	160:
		IF NOT DP_SinStepe THEN	
				IF arrAxisCtrl[AxiseNo.AxisName.AnDTCarryingUpDown].Status.Homed AND arrAxisCtrl[AxiseNo.AxisName.AnDTCarryingUpDown].Status.NoMoving AND 
					NOT arrAxisCtrl[AxiseNo.AxisName.AnDTCarryingUpDown].Status.Error AND arrAxisCtrl[AxiseNo.AxisName.AnDTCarryingLine].Cmd.arrbRealPoint[1] THEN
							IF arrAxisCtrl[AxiseNo.AxisName.AnDTCarryingUpDown].Cmd.arrbRealPoint[2] THEN
								arrAxisCtrl[AxiseNo.AxisName.AnDTCarryingUpDown].Cmd.iGoSetPos:=0;
							ELSE
								arrAxisCtrl[AxiseNo.AxisName.AnDTCarryingUpDown].Cmd.iGoSetPos:=2;//正极叠片平台升降去取片位 放片
							END_IF
				END_IF
				IF 	arrAxisCtrl[AxiseNo.AxisName.AnDTCarryingUpDown].Cmd.arrbRealPoint[2] AND arrAxisCtrl[AxiseNo.AxisName.AnDTCarryingUpDown].Status.Homed THEN
								IF Mach_Control.DT_b.SinStepMode THEN//单步调试模式
									DP_SinStepe:=TRUE;
								ELSE
									DP_SinStepe:=FALSE;	
								END_IF				
								An_Step2:=170;
				END_IF	
		END_IF
	
	170:

			arrCyCtrl[arrCyNo.ElectValveName.AnDTCarryingVacuum].Cmd.bOFF:=FALSE;//正极叠片搬运真空关
			arrCyCtrl[arrCyNo.ElectValveName.AnDTCarryingVacuum].Cmd.bON:=TRUE;//正极叠片搬运真空关
			arrCyCtrl[arrCyNo.ElectValveName.AnDTCarryingVacuumBark].Cmd.bON:=TRUE;//正极叠片搬运破真空开
			arrCyCtrl[arrCyNo.ElectValveName.AnDTCarryingVacuumBark].Cmd.bOFF:=FALSE;//正极叠片搬运破真空开
			arrCyCtrl[arrCyNo.ElectValveName.AndeviationVacuum].Cmd.bON:=TRUE;//正极纠偏平台真空开		
			arrCyCtrl[arrCyNo.ElectValveName.AndeviationVacuum].Cmd.bOFF:=FALSE;//正极纠偏平台真空开	
			//IF Mach_Control.An_b.An_DPCarryingFalg THEN	
				Mach_Control.An_b.An_DPCarryingFalg :=FALSE;//复位正极叠片搬运吸盘上有料标记
				Mach_Control.An_b.An_deviationFalg:=TRUE;//置位纠偏平台上有料标记
			//END_IF
			An_Step2:=180;

			
	180:
		IF NOT DP_SinStepe THEN	
				IF arrAxisCtrl[AxiseNo.AxisName.AnDTCarryingUpDown].Status.Homed AND arrAxisCtrl[AxiseNo.AxisName.AnDTCarryingUpDown].Status.NoMoving AND 
					NOT arrAxisCtrl[AxiseNo.AxisName.AnDTCarryingUpDown].Status.Error AND arrAxisCtrl[AxiseNo.AxisName.AnDTCarryingLine].Cmd.arrbRealPoint[1] THEN
							IF arrAxisCtrl[AxiseNo.AxisName.AnDTCarryingUpDown].Cmd.arrbRealPoint[4] THEN
								arrAxisCtrl[AxiseNo.AxisName.AnDTCarryingUpDown].Cmd.iGoSetPos:=0;
							ELSE
								arrAxisCtrl[AxiseNo.AxisName.AnDTCarryingUpDown].Cmd.iGoSetPos:=4;//正极叠片平台升降去等待位
							END_IF
				END_IF
				IF 	arrAxisCtrl[AxiseNo.AxisName.AnDTCarryingUpDown].Cmd.arrbRealPoint[4] AND arrAxisCtrl[AxiseNo.AxisName.AnDTCarryingUpDown].Status.Homed THEN
								IF Mach_Control.DT_b.SinStepMode THEN//单步调试模式
									DP_SinStepe:=TRUE;
								ELSE
									DP_SinStepe:=FALSE;	
								END_IF				
								An_Step2:=190;
				END_IF	
		END_IF	
	190:
			YS.IN:=TRUE;
			
		IF 	 (Mach_Control.An_b.RectifydevDone OR CCD.AnRec.Finish.RectifyResult=2 OR CCD.AnRec.Finish.RectifyResult=3 OR CCD.AnRec.Finish.RectifyResult=4) AND YS.Q  THEN
			Mach_Control.An_b.An_Rectifydev_CS:=Mach_Control.An_b.An_Rectifydev_CS+1;
			An_Step2:=200;
			YS.IN:=FALSE;
		END_IF
		
	200:
		IF NOT DP_SinStepe THEN	
				IF arrAxisCtrl[AxiseNo.AxisName.AnDTCarryingUpDown].Status.Homed AND arrAxisCtrl[AxiseNo.AxisName.AnDTCarryingUpDown].Status.NoMoving AND 
					NOT arrAxisCtrl[AxiseNo.AxisName.AnDTCarryingUpDown].Status.Error AND arrAxisCtrl[AxiseNo.AxisName.AnDTCarryingLine].Cmd.arrbRealPoint[1] THEN
							IF arrAxisCtrl[AxiseNo.AxisName.AnDTCarryingUpDown].Cmd.arrbRealPoint[2] THEN
								arrAxisCtrl[AxiseNo.AxisName.AnDTCarryingUpDown].Cmd.iGoSetPos:=0;
							ELSE
								arrAxisCtrl[AxiseNo.AxisName.AnDTCarryingUpDown].Cmd.iGoSetPos:=2;//正极叠片平台升降去取片位 放片
							END_IF
				END_IF
				IF 	arrAxisCtrl[AxiseNo.AxisName.AnDTCarryingUpDown].Cmd.arrbRealPoint[2] AND arrAxisCtrl[AxiseNo.AxisName.AnDTCarryingUpDown].Status.Homed THEN
								IF Mach_Control.DT_b.SinStepMode THEN//单步调试模式
									DP_SinStepe:=TRUE;
								ELSE
									DP_SinStepe:=FALSE;	
								END_IF				
								An_Step2:=220;
								IF Mach_Control.DT_b.DT_CCD_TwoModel THEN												
										CCD.AnRec.Finish.RectifyResult:=0;
										CCD.AnRec.Finish.RectifyX1:=0;
										CCD.AnRec.Finish.RectifyX2:=0;
										CCD.AnRec.Finish.RectifyY:=0;												
										Mach_Control.An_b.An_CCDStart :=TRUE;//启动CCD拍照
										CCD.AnRec.Start.iPhotoDo:=2;//第二次拍照		
								END_IF	
				END_IF	
		END_IF	
		
			
	220:
	
			arrCyCtrl[arrCyNo.ElectValveName.AnDTCarryingVacuum].Cmd.bON:=FALSE;//正极叠片搬运真空开
			arrCyCtrl[arrCyNo.ElectValveName.AnDTCarryingVacuum].Cmd.bOFF:=TRUE;//正极叠片搬运真空开
			arrCyCtrl[arrCyNo.ElectValveName.AnDTCarryingVacuumBark].Cmd.bOFF:=TRUE;//正极叠片搬运破真空关
			arrCyCtrl[arrCyNo.ElectValveName.AnDTCarryingVacuumBark].Cmd.bON:=FALSE;//正极叠片搬运破真空关
			arrCyCtrl[arrCyNo.ElectValveName.AndeviationVacuum].Cmd.bOFF:=TRUE;//正极纠偏平台真空关	
			arrCyCtrl[arrCyNo.ElectValveName.AndeviationVacuum].Cmd.bON:=FALSE;//正极纠偏平台真空关	
			arrCyCtrl[arrCyNo.ElectValveName.AndeviationVacuumBark].Cmd.bON:=TRUE;//正极纠偏平台破真空开	
			arrCyCtrl[arrCyNo.ElectValveName.AndeviationVacuumBark].Cmd.bOFF:=FALSE;//正极纠偏平台破真空开	
			//IF Mach_Control.An_b.An_deviationFalg THEN
				Mach_Control.An_b.An_DPCarryingFalg :=TRUE;//叠片搬运吸盘上有料标记
				Mach_Control.An_b.An_deviationFalg:=FALSE;//纠偏平台上有料标记
			//END_IF
			YS1.IN:=TRUE;
			IF YS1.Q THEN
			An_Step2:=230;
			YS1.IN:=FALSE;
			END_IF
	
	
	230:
		IF NOT DP_SinStepe THEN	
				IF arrAxisCtrl[AxiseNo.AxisName.AnDTCarryingUpDown].Status.Homed AND arrAxisCtrl[AxiseNo.AxisName.AnDTCarryingUpDown].Status.NoMoving AND 
					NOT arrAxisCtrl[AxiseNo.AxisName.AnDTCarryingUpDown].Status.Error AND arrAxisCtrl[AxiseNo.AxisName.AnDTCarryingLine].Cmd.arrbRealPoint[1] THEN
							IF arrAxisCtrl[AxiseNo.AxisName.AnDTCarryingUpDown].Cmd.arrbRealPoint[4] THEN
								arrAxisCtrl[AxiseNo.AxisName.AnDTCarryingUpDown].Cmd.iGoSetPos:=0;
							ELSE
								arrAxisCtrl[AxiseNo.AxisName.AnDTCarryingUpDown].Cmd.iGoSetPos:=4;//正极叠片平台升降去等待位
							END_IF
				END_IF
				IF 	arrAxisCtrl[AxiseNo.AxisName.AnDTCarryingUpDown].Cmd.arrbRealPoint[4] AND arrAxisCtrl[AxiseNo.AxisName.AnDTCarryingUpDown].Status.Homed THEN
								IF Mach_Control.DT_b.SinStepMode THEN//单步调试模式
									DP_SinStepe:=TRUE;
								ELSE
									DP_SinStepe:=FALSE;	
								END_IF				
								An_Step2:=6666;
				END_IF	
		END_IF	
	
	
		
			
		
		
END_CASE
END_IF
END_ACTION

ACTION An_StandbySub4:
IF Mach_Control.U.DT_iMode=1 THEN//在自动状态下	
//An_Step3----正极叠片搬运取纠偏极片
CASE An_Step3 OF
	10://正极NG料盒气缸伸出	
		IF  arrAxisCtrl[AxiseNo.AxisName.AnDTCarryingUpDown].Status.Enabled AND  arrAxisCtrl[AxiseNo.AxisName.AnDTCarryingLine].Status.Enabled THEN	
			arrCyCtrl[arrCyNo.CylinderName.AnScrapbinCy].Cmd.bON:=TRUE;//正极纠偏气缸伸出
			IF  arrCyCtrl[arrCyNo.CylinderName.AnScrapbinCy].Status.ONState THEN
				An_Step3:=11;
			END_IF
		END_IF
	11://正极叠片搬运升降至等待位		
					IF NOT DP_SinStepe THEN	
						(*
						IF arrAxisCtrl[AxiseNo.AxisName.AnCarryingUpDown].Status.Homed AND arrAxisCtrl[AxiseNo.AxisName.AnCarryingUpDown].Status.NoMoving AND 
							NOT arrAxisCtrl[AxiseNo.AxisName.AnCarryingUpDown].Status.Error THEN
									IF arrAxisCtrl[AxiseNo.AxisName.AnCarryingUpDown].Cmd.arrbRealPoint[4] THEN
										arrAxisCtrl[AxiseNo.AxisName.AnCarryingUpDown].Cmd.iGoSetPos:=0;
									ELSE
										arrAxisCtrl[AxiseNo.AxisName.AnCarryingUpDown].Cmd.iGoSetPos:=4;//正极送片搬运升降等待高度
									END_IF
						END_IF
						*)
						IF arrAxisCtrl[AxiseNo.AxisName.AnDTCarryingUpDown].Status.Homed AND arrAxisCtrl[AxiseNo.AxisName.AnDTCarryingUpDown].Status.NoMoving AND 
							NOT arrAxisCtrl[AxiseNo.AxisName.AnDTCarryingUpDown].Status.Error THEN
									IF arrAxisCtrl[AxiseNo.AxisName.AnDTCarryingUpDown].Cmd.arrbRealPoint[4] THEN
										arrAxisCtrl[AxiseNo.AxisName.AnDTCarryingUpDown].Cmd.iGoSetPos:=0;
									ELSE
										arrAxisCtrl[AxiseNo.AxisName.AnDTCarryingUpDown].Cmd.iGoSetPos:=4;//正极叠片平台升降至等待高度
									END_IF
						END_IF
						IF 	arrAxisCtrl[AxiseNo.AxisName.AnDTCarryingUpDown].Cmd.arrbRealPoint[4] AND arrAxisCtrl[AxiseNo.AxisName.AnDTCarryingUpDown].Status.Homed THEN
										IF Mach_Control.DT_b.SinStepMode THEN//单步调试模式
											DP_SinStepe:=TRUE;
										ELSE
											DP_SinStepe:=FALSE;	
										END_IF				
										An_Step3:=30;
						END_IF	
				END_IF								
	20://正极搬运平移回初始位
		IF NOT DP_SinStepe THEN
				IF arrAxisCtrl[AxiseNo.AxisName.AnCarryingUpDown].Cmd.arrbRealPoint[4] AND arrAxisCtrl[AxiseNo.AxisName.AnCarryingLine].Status.Homed AND
					 arrAxisCtrl[AxiseNo.AxisName.AnCarryingLine].Status.NoMoving AND NOT arrAxisCtrl[AxiseNo.AxisName.AnCarryingLine].Status.Error THEN
							IF arrAxisCtrl[AxiseNo.AxisName.AnCarryingLine].Cmd.arrbRealPoint[1] THEN
									An_CarryingTorMark:=FALSE;//正极搬运1移位力矩判断标志位
									arrAxisCtrl[AxiseNo.AxisName.AnCarryingLine].Cmd.iGoSetPos:=0;
									IF Mach_Control.DT_b.SinStepMode THEN//单步调试模式
										DP_SinStepe:=TRUE;
									ELSE
										DP_SinStepe:=FALSE;	
									END_IF	
									An_Step3:=30;
							ELSE
								arrAxisCtrl[AxiseNo.AxisName.AnCarryingLine].Cmd.iGoSetPos:=1;//正极搬运平移到初始位
								An_CarryingTorMark:=TRUE;//正极搬运1移位力矩判断标志位
							END_IF
				END_IF	
		END_IF
	30://正极叠片搬运平移至初始位，
			//IF arrAxisCtrl[AxiseNo.AxisName.AnDTCarryingLine].Status.fActPos < (arrAxisPar[AxiseNo.AxisName.AnDTCarryingLine].arrTargetPoint[2]-180) THEN
	          //arrCyCtrl[arrCyNo.ElectValveName.AndeviationIonizedWind].Cmd.bON:=TRUE;//正极纠偏平台除尘
			   //arrCyCtrl[arrCyNo.ElectValveName.AndeviationIonizedWind].Cmd.bOff:=FALSE;//正极纠偏平台除尘
	      // END_IF
			IF NOT DP_SinStepe THEN
						arrCyCtrl[arrCyNo.CylinderName.AnScrapbinCy].Cmd.bON:=TRUE;//正极纠偏气缸伸出
						IF   arrAxisCtrl[AxiseNo.AxisName.AnDTCarryingUpDown].Cmd.arrbRealPoint[4] AND arrAxisCtrl[AxiseNo.AxisName.AnDTCarryingLine].Status.Homed AND
							 arrAxisCtrl[AxiseNo.AxisName.AnDTCarryingLine].Status.NoMoving AND NOT arrAxisCtrl[AxiseNo.AxisName.AnDTCarryingLine].Status.Error  AND 
							 NOT arrAxisCtrl[AxiseNo.AxisName.AnCarryingLine].Status.Error 
                             AND LREAL_TO_REAL(arrAxisCtrl[AxiseNo.AxisName.AnCarryingLine].Status.fActPos) < (arrAxisPar[AxiseNo.AxisName.AnCarryingLine].arrTargetPoint[2]-50) AND
							 arrCyCtrl[arrCyNo.CylinderName.AnScrapbinCy].Status.ONState THEN
									IF arrAxisCtrl[AxiseNo.AxisName.AnDTCarryingLine].Cmd.arrbRealPoint[1] THEN
										An_DTCarryingTorMark:=FALSE;//正极叠台搬运力矩判断标志位
										arrAxisCtrl[AxiseNo.AxisName.AnDTCarryingLine].Cmd.iGoSetPos:=0;
										IF Mach_Control.DT_b.SinStepMode THEN//单步调试模式
											DP_SinStepe:=TRUE;
										ELSE
											DP_SinStepe:=FALSE;	
										END_IF								
										An_Step3:=40;
									ELSE
										arrAxisCtrl[AxiseNo.AxisName.AnDTCarryingLine].Cmd.iGoSetPos:=1;//正极叠片平移移动至初始位
										An_DTCarryingTorMark:=TRUE;//正极叠台搬运力矩判断标志位
									END_IF
						END_IF
			END_IF
	40://判断纠偏平台是否允许取极片
			IF NOT DP_SinStepe THEN
					IF Mach_Control.An_b.An_deviationDPOK OR Mach_Control.U.EmptyRunMode THEN
						IF Mach_Control.DT_b.SinStepMode THEN//单步调试模式
							DP_SinStepe:=TRUE;
						ELSE
							DP_SinStepe:=FALSE;	
						END_IF			
					//	CCD正极纠偏平台二次拍照-------------复检拍照
						IF Mach_Control.DT_b.DT_CCD_TwoModel THEN												
							CCD.AnRec.Finish.RectifyResult:=0;
							CCD.AnRec.Finish.RectifyX1:=0;
							CCD.AnRec.Finish.RectifyX2:=0;
							CCD.AnRec.Finish.RectifyY:=0;												
							Mach_Control.An_b.An_CCDStart :=TRUE;//启动CCD拍照
							CCD.AnRec.Start.iPhotoDo:=2;//第二次拍照		
						END_IF	
						An_TON[6].IN:=FALSE;
						An_Step3:=50;
					END_IF
			END_IF
END_CASE
END_IF


CASE An_Step3 OF
	50://AND arrCyCtrl[arrCyNo.CylinderName.AnScrapbinCy].Io.DIOnSwitch
		IF NOT DP_SinStepe THEN
			arrCyCtrl[arrCyNo.ElectValveName.AnDTCarryingVacuum].Cmd.bON:=FALSE;//正极叠片搬运升降真空开
			arrCyCtrl[arrCyNo.ElectValveName.AnDTCarryingVacuum].Cmd.bOFF:=TRUE;//正极叠片搬运真空开
			IF arrAxisCtrl[AxiseNo.AxisName.AnDTCarryingUpDown].Status.Homed AND arrAxisCtrl[AxiseNo.AxisName.AnDTCarryingUpDown].Status.NoMoving AND 
			NOT arrAxisCtrl[AxiseNo.AxisName.AnDTCarryingUpDown].Status.Error  THEN
				IF arrAxisCtrl[AxiseNo.AxisName.AnDTCarryingUpDown].Cmd.arrbRealPoint[2] THEN
					arrCyCtrl[arrCyNo.ElectValveName.AndeviationVacuum].Cmd.bOFF:=TRUE;//正极纠偏真空关
					arrCyCtrl[arrCyNo.ElectValveName.AndeviationVacuum].Cmd.bON:=FALSE;//正极纠偏真空关
					arrCyCtrl[arrCyNo.ElectValveName.AndeviationVacuumBark].Cmd.bON:=TRUE;//正极纠偏破真空开
					arrCyCtrl[arrCyNo.ElectValveName.AndeviationVacuumBark].Cmd.bOFF:=FALSE;//正极纠偏破真空开
					arrAxisCtrl[AxiseNo.AxisName.AnDTCarryingUpDown].Cmd.iGoSetPos:=0;
					//IF Mach_Control.An_b.An_deviationFalg THEN
						Mach_Control.An_b.An_DPCarryingFalg:=TRUE;// 复位正极叠片搬运真空吸盘标记有料
						Mach_Control.An_b.An_deviationFalg:=FALSE;//复位正极纠偏平台有料标记	
					//END_IF
					Par.stDT_date.An_MQ_Slice[2]:=Par.stDT_date.An_MQ_Slice[1];												
																
					IF NOT An_TON[6].Q THEN
						An_TON[6].IN:=TRUE;
					ELSE
						IF Mach_Control.DT_b.SinStepMode THEN//单步调试模式
							DP_SinStepe:=TRUE;
						ELSE
							DP_SinStepe:=FALSE;	
						END_IF		
						An_TON[6].IN:=FALSE;				
						An_Step3:=60;											
					END_IF									
				ELSE
					arrAxisCtrl[AxiseNo.AxisName.AnDTCarryingUpDown].Cmd.iGoSetPos:=2;//正极叠片平台升降下降至取料高度
				END_IF
			
			END_IF	
		END_IF
	60://正极叠片搬运升降上升至初始位
		IF arrAxisCtrl[AxiseNo.AxisName.AnDTCarryingUpDown].Status.Homed AND arrAxisCtrl[AxiseNo.AxisName.AnDTCarryingUpDown].Status.NoMoving AND 
		NOT arrAxisCtrl[AxiseNo.AxisName.AnDTCarryingUpDown].Status.Error THEN
			IF arrAxisCtrl[AxiseNo.AxisName.AnDTCarryingUpDown].Cmd.arrbRealPoint[4] THEN
				arrAxisCtrl[AxiseNo.AxisName.AnDTCarryingUpDown].Cmd.iGoSetPos:=0;
				An_Step3:=6666;
			ELSE
				arrAxisCtrl[AxiseNo.AxisName.AnDTCarryingUpDown].Cmd.iGoSetPos:=4;//正极叠片平台升降上升至初始位
			END_IF
		END_IF		
END_CASE
END_ACTION

ACTION Ca_Alarm:
//报警延时时间
Ca_AlarmTON[1](IN:= , PT:=T#80MS , Q=> , ET=> );//负极取流水线搬运升降机械手吸盘误吸极片报警延时
Ca_AlarmTON[2](IN:= , PT:=T#80MS , Q=> , ET=> );//负极取流水线搬运升降机械手吸盘掉片报警延时
Ca_AlarmTON[3](IN:= , PT:=T#80MS , Q=> , ET=> );///负极送片搬运升降机械手误吸极片报警延时
Ca_AlarmTON[4](IN:= , PT:=T#80MS , Q=> , ET=> );////负极取流水线搬运升降机械手吸盘掉片	报警延时
Ca_AlarmTON[5](IN:= , PT:=T#80MS , Q=> , ET=> );///负极叠台搬运升降机械手误吸极片报警延时
Ca_AlarmTON[6](IN:= , PT:=T#80MS , Q=> , ET=> );////负极叠台搬运升降机械手吸盘掉片报警延时
Ca_AlarmTON[7](IN:= , PT:=T#80MS , Q=> , ET=> );///负极纠偏平台误吸极片报警延时
Ca_AlarmTON[8](IN:= , PT:=T#150MS , Q=> , ET=> );////负极纠偏平台吸盘掉片报警延时
Ca_AlarmTON[9](IN:= , PT:=T#300MS , Q=> , ET=> );
Ca_AlarmTON[10](IN:= , PT:=T#300MS , Q=> , ET=> );
Ca_AlarmTON[11](IN:= , PT:=T#300MS , Q=> , ET=> );//负极极片对齐度检测返回结果超时
Ca_AlarmTon[12](IN:= , PT:=T#400MS , Q=> , ET=> );//负极CCD纠偏平台检测返回结果超时
Ca_AlarmTon[13](IN:=CaCCDMark , PT:=T#50MS , Q=> , ET=> );//负极CCD纠偏平台检测返回结果超时
Ca_AlarmTon[15](IN:= , PT:=T#50MS , Q=> , ET=> );//负极取片搬运叠片过程中的真空处理
Ca_AlarmTon[16](IN:= , PT:=T#50MS , Q=> , ET=> );//负极取片搬运叠片过程中的真空处理
Ca_AlarmTon[17](IN:=NOT Mach_Control.se.CaNGboxsensor , PT:=T#5S , Q=> , ET=> );//负极NG料盒料满	

rCaUse[1](CLK:=Ca_Step0=40, Q=> );
rCaUse[2](CLK:=Mach_Control.Ca_b.Ca_CCDStart AND NOT   Mach_Control.Ca_b.Demarcateing , Q=> );
rCaUse[3](CLK:=Par.stDT_date.Ca_Rectifydev_Btn , Q=> );
rCaUse[4](CLK:= NOT arrCyCtrl[arrCyNo.ElectValveName.CaCarryingVacuum2].Io.DOStatus1 , Q=> ); 
rCaUse[5](CLK:= NOT arrCyCtrl[arrCyNo.ElectValveName.CaDTCarryingVacuum].Io.DOStatus1 , Q=> );
rCaUse[6](CLK:=arrCyCtrl[arrCyNo.ElectValveName.CaCarryingVacuum1].Io.DOStatus1 , Q=> ); 

//Mach_Control.Ca_b.Error[1]:=TRUE;//负极取流水线搬运升降有真空信号，无极片报警
//Mach_Control.Ca_b.Error[2]:=TRUE;//负极取流水线搬运升降有极片，无真空信号报警
//Mach_Control.Ca_b.Error[3]:=TRUE;//负极送片搬运升降有真空信号，无极片报警
//Mach_Control.Ca_b.Error[4]:=TRUE;//负极送片搬运升降取片过程中真空报警,有极片，无真空信号
//Mach_Control.Ca_b.Error[5]:=TRUE;//负极叠台搬运升降有真空信号，无极片报警
//Mach_Control.Ca_b.Error[6]:=TRUE;//负极叠台搬运升降有极片，无真空信号报警
//Mach_Control.Ca_b.Error[7]:=TRUE;//纠偏平台无片极，有真空信号报警
//Mach_Control.Ca_b.Error[8]:=TRUE;//纠偏平台有极片，无真空报警
//Mach_Control.Ca_b.Error[9]:=TRUE;//纠偏CCD拍照完成IO信号未给出
//Mach_Control.Ca_b.Error[10] //CCD标定NG报警
//Mach_Control.Ca_b.Error[11]:=TRUE;//负极藕合凸轮报警
//Mach_Control.Ca_b.Error[12]:=TRUE;//负极NG收纳盒满料报警
//Mach_Control.Ca_b.Error[13];
//Mach_Control.Ca_b.Error[14];
//Mach_Control.Ca_b.Error[15];
//Mach_Control.Ca_b.Error[16];
//Mach_Control.Ca_b.Error[17]:=TRUE;//负极防撞感应信报警
//Mach_Control.Ca_b.Error[18] :=TRUE;//负极CCD纠偏平台检测返回结果超时
//Mach_Control.Ca_b.Error[19]:=TRUE;//负极取放料回原点超时报警
//Mach_Control.Ca_b.Error[20]:=TRUE;//负极皮带回原点超时报警	
//Mach_Control.Ca_b.Error[21]:=TRUE;//负极纠偏平台连续NG报警
//Mach_Control.Ca_b.Error[22]:=TRUE;//负极叠台搬运升降真空报警，电芯上有片，请拿掉
//Mach_Control.Ca_b.Error[23]:=TRUE;//负极叠台搬运升降真空报警，电芯上无掉片
//Mach_Control.Ca_b.Error[24] //负极纠偏平台NG片未排掉报警，请拿掉
//Mach_Control.Ca_b.Error[25] //负极极片对齐度检测返回结果超时
//Mach_Control.Ca_b.Error[26]:=TRUE;//负极搬运平移防撞软限位报警
//Mach_Control.Ca_b.Error[27] ////负极极片对齐度检测返回结果无片报警
//Mach_Control.Ca_b.Error[28] //负极极片NG料盒料满
//Mach_Control.Ca_b.Error[29]:=TRUE;	  //负极初始化时负极叠片搬运升降吸盘有真空报警
//Mach_Control.Ca_b.Error[30]:=TRUE;	  //负极初始化时负极送片搬运升降2吸盘有真空报警
//Mach_Control.Ca_b.Error[31]:=TRUE;	   //负极皮带初始化时负极送片搬运升降1吸盘有真空报警


//Mach_Control.Ca_b.Error[32]:=TRUE;//负极取片叠片过程中真空报警
//Mach_Control.Ca_b.Error[33]:=TRUE;//纠偏平台有片，请拿走
//Mach_Control.Ca_b.Error[34]:=TRUE;//负极叠台搬运平移取片时真空报警
//Mach_Control.Ca_b.Error[35]:=TRUE;//负极纠偏台NG料盒料满报警
//Mach_Control.Ca_b.Error[36]:=TRUE;//负极纠偏纠偏CCD返回结果超时
//Mach_Control.Ca_b.Error[38] :=TRUE;//负极叠台搬运升降有极耳无真空报警
//Mach_Control.Ca_b.Error[39] :=TRUE;//负极叠台搬运升降有极耳无真空报警
//Mach_Control.Ca_b.Error[40] S=AnOverNGcount>=3;//负极单张踢废连续NG
//Mach_Control.Ca_b.Error[41] :=TRUE;//负极缓存皮带准备运动时，负极升降1不在安全位报警
//Mach_Control.Ca_b.Error[42] :=TRUE;//负极机械手初始化时，叠台搬运升降不在避让位
Mach_Control.Ca_b.Error[40] S=CaOverNGcount>=3;//负极单张踢废连续NG

//NG料盒料满报警
	IF (*Par.stDT_date.Ca_Rectifydev_JS>=Par.stDT_date.Ca_Rectifydev_NGSet OR*) Ca_AlarmTon[17].Q THEN
		Mach_Control.Ca_b.Error[35]:=TRUE;//负极纠偏台NG料盒料满报警
	ELSE
		Mach_Control.Ca_b.Error[35]:=FALSE;//负极纠偏台NG料盒料满报警
	END_IF
	IF rCaUse[3].Q THEN
		Par.stDT_date.Ca_Rectifydev_JS:=0;
	END_IF
	
	
	
//负极初始化时有真空报警	
	IF Mach_Control.Ca_b.Ca_GohomeHMI  THEN
			IF  arrCyCtrl[arrCyNo.ElectValveName.CaDTCarryingVacuum].Status.ONState  THEN
				Mach_Control.Ca_b.Error[29]:=TRUE;	  //负极初始化时负极叠片搬运升降吸盘有真空报警
			END_IF
			IF arrCyCtrl[arrCyNo.ElectValveName.CaCarryingVacuum2].Status.ONState THEN
				Mach_Control.Ca_b.Error[30]:=TRUE;	  //负极初始化时负极送片搬运升降2吸盘有真空报警
			END_IF
	END_IF	
//负极皮带初始化时有真空报警	
	IF Mach_Control.Ca_b.Ca_BeltGohomeHMI  AND arrCyCtrl[arrCyNo.ElectValveName.CaCarryingVacuum1].Status.ONState THEN
		Mach_Control.Ca_b.Error[31]:=TRUE;	   //负极皮带初始化时负极送片搬运升降1吸盘有真空报警
	END_IF	
	
//负极取流水线搬运机械手升降吸盘真空信号与搬运升降极片有无料标记不一致报警
Ca_AlarmTON[1].IN:=NOT arrCyCtrl[arrCyNo.ElectValveName.CaCarryingVacuum1].Io.DOStatus1 AND  arrCyCtrl[arrCyNo.ElectValveName.CaCarryingVacuum1].Io.DIOnSwitch 
	AND NOT Mach_Control.Ca_b.Ca_SegbeltFalg AND NOT Mach_Control.U.EmptyRunMode AND  Mach_Control.U.DT_iMode=1 AND NOT Mach_Control.Ca_b.Error[2] ;
rtVacALM[1](CLK:=Ca_AlarmTON[1].Q, Q=> );		
		IF  rtVacALM[1].Q THEN
			//Mach_Control.Ca_b.Ca_SegbeltFalg:=FALSE;
			Mach_Control.Ca_b.Error[1]:=TRUE;//负极取流水线搬运升降有真空信号，无极片报警
		END_IF

//
Ca_AlarmTON[2].IN:=NOT arrCyCtrl[arrCyNo.ElectValveName.CaCarryingVacuum1].Io.DIOnSwitch AND  Mach_Control.Ca_b.Ca_SegbeltFalg AND NOT Mach_Control.U.EmptyRunMode AND
	arrAxisCtrl[AxiseNo.AxisName.CaCarryingUpDown1].Status.fActPos<=(arrAxisPar[AxiseNo.AxisName.CaCarryingUpDown1].arrTargetPoint[2]-5) AND arrCyCtrl[arrCyNo.ElectValveName.CaCarryingVacuum1].Io.DOStatus1 ;		
rtVacALM[2](CLK:=Ca_AlarmTON[2].Q, Q=> );	
		IF  rtVacALM[2].Q THEN
			Mach_Control.Ca_b.Error[2]:=TRUE;//负极取流水线搬运升降有极片，无真空信号报警
		END_IF	
	
(*
//负极取流水线搬运机械手升降吸盘真空信号与搬运升降极片有无料标记不一致报警
Ca_AlarmTON[1].IN:=NOT arrCyCtrl[arrCyNo.ElectValveName.CaCarryingVacuum1].Io.DOStatus1 AND  arrCyCtrl[arrCyNo.ElectValveName.CaCarryingVacuum1].Io.DIOnSwitch 
	AND NOT Mach_Control.Ca_b.Ca_SegbeltFalg AND NOT Mach_Control.U.EmptyRunMode AND  Mach_Control.U.DT_iMode=1 AND NOT Mach_Control.Ca_b.Error[2] ;
		IF  Ca_AlarmTON[1].Q THEN
			//Mach_Control.Ca_b.Ca_SegbeltFalg:=FALSE;
			Mach_Control.Ca_b.Error[1]:=TRUE;//负极取流水线搬运升降有真空信号，无极片报警
		END_IF

//
Ca_AlarmTON[2].IN:=NOT arrCyCtrl[arrCyNo.ElectValveName.CaCarryingVacuum1].Io.DIOnSwitch AND  Mach_Control.Ca_b.Ca_SegbeltFalg AND NOT Mach_Control.U.EmptyRunMode AND
	arrAxisCtrl[AxiseNo.AxisName.CaCarryingUpDown1].Status.fActPos<=(arrAxisPar[AxiseNo.AxisName.CaCarryingUpDown1].arrTargetPoint[2]-5) AND arrCyCtrl[arrCyNo.ElectValveName.CaCarryingVacuum1].Io.DOStatus1 ;		
		IF  Ca_AlarmTON[2].Q THEN
			(*
			arrCyCtrl[arrCyNo.ElectValveName.CaCarryingVacuum1]	.Cmd.bOFF:=TRUE;//负极搬运1真空关
			arrCyCtrl[arrCyNo.ElectValveName.CaCarryingVacuum1]	.Cmd.bON:=FALSE;//负极搬运1真空开
			arrCyCtrl[arrCyNo.ElectValveName.CaCarryingVacuumBark1]	.Cmd.bOFF:=FALSE;//负极搬运1真空关
			arrCyCtrl[arrCyNo.ElectValveName.CaCarryingVacuumBark1]	.Cmd.bON:=TRUE;//负极搬运1真空开
			Mach_Control.Ca_b.Ca_SegbeltFalg:=FALSE;
			*)
			Mach_Control.Ca_b.Error[2]:=TRUE;//负极取流水线搬运升降有极片，无真空信号报警
		END_IF
IF Mach_Control.Ca_b.Error[2] AND arrCyCtrl[arrCyNo.ElectValveName.CaCarryingVacuum1].Io.DIOnSwitch AND rCa_AlarmReset.Q  THEN
	Mach_Control.Ca_b.Error[2]:=FALSE;//负极取流水线搬运升降有极片，无真空信号报警
ELSIF Mach_Control.Ca_b.Error[2] AND NOT arrCyCtrl[arrCyNo.ElectValveName.CaCarryingVacuum1].Io.DIOnSwitch AND rCa_AlarmReset.Q  THEN
	arrCyCtrl[arrCyNo.ElectValveName.CaCarryingVacuum1]	.Cmd.bOFF:=TRUE;//负极搬运1真空关
	arrCyCtrl[arrCyNo.ElectValveName.CaCarryingVacuum1]	.Cmd.bON:=FALSE;//负极搬运1真空开
	arrCyCtrl[arrCyNo.ElectValveName.CaCarryingVacuumBark1]	.Cmd.bOFF:=FALSE;//负极搬运1真空关
	arrCyCtrl[arrCyNo.ElectValveName.CaCarryingVacuumBark1]	.Cmd.bON:=TRUE;//负极搬运1真空开
	Ca_StandbyStep2:=0;
	Mach_Control.Ca_b.Ca_SegbeltFalg:=FALSE;
	Mach_Control.Ca_b.Error[2]:=FALSE;//负极取流水线搬运升降有极片，无真空信号报警
END_IF
*)		

//负极取片搬运取片过程中的真空报警处理
Ca_AlarmTON[4].IN:=NOT arrCyCtrl[arrCyNo.ElectValveName.CaCarryingVacuum2].Io.DIOnSwitch AND Mach_Control.Ca_b.Ca_CarryingFalg 
	AND NOT Mach_Control.U.EmptyRunMode AND arrAxisCtrl[AxiseNo.AxisName.CaCarryingUpDown2].Status.Homed 
	AND arrAxisCtrl[AxiseNo.AxisName.CaCarryingUpDown2].Status.fActPos<=(arrAxisPar[AxiseNo.AxisName.CaCarryingUpDown2].arrTargetPoint[2]-5)//AND NOT Blueflaging
	AND NOT  arrCyCtrl[arrCyNo.ElectValveName.CaCarryingVacuum2].Io.DOStatus1 AND NOT Bnt_Blueflaging  AND  arrAxisCtrl[AxiseNo.AxisName.CaCarryingLine2].Status.NoMoving ;
		IF  Ca_AlarmTON[4].Q THEN  
				Mach_Control.Ca_b.Error[4]:=TRUE;//负极送片搬运升降机械有极片，无真空信号报警
				(*
				Mach_Control.Ca_b.Ca_CarryingFalg :=FALSE;
				arrCyCtrl[arrCyNo.ElectValveName.CaCarryingVacuum2]	.Cmd.bON:=TRUE;//负极搬运2真空破
				arrCyCtrl[arrCyNo.ElectValveName.CaCarryingVacuum2]	.Cmd.bOFF:=FALSE;//负极搬运2真空破
				*)
		END_IF
IF Mach_Control.Ca_b.Error[4] AND arrCyCtrl[arrCyNo.ElectValveName.CaCarryingVacuum2].Io.DIOnSwitch AND rCa_AlarmReset.Q  THEN
	Mach_Control.Ca_b.Error[4]:=FALSE;//负极送片搬运升降机械有极片，无真空信号报警
ELSIF Mach_Control.Ca_b.Error[4] AND NOT arrCyCtrl[arrCyNo.ElectValveName.CaCarryingVacuum2].Io.DIOnSwitch AND rCa_AlarmReset.Q  THEN
	arrCyCtrl[arrCyNo.ElectValveName.CaCarryingVacuum2]	.Cmd.bON:=TRUE;//负极搬运2真空破
	arrCyCtrl[arrCyNo.ElectValveName.CaCarryingVacuum2]	.Cmd.bOFF:=FALSE;//负极搬运2真空破
	Ca_StandbyStep0:=0;
	Ca_Step0:=0;
	Ca_Step1:=0;
	Ca_Step2:=0;
	Ca_Step3:=0;
	Mach_Control.Ca_b.Error[4]:=FALSE;//负极送片搬运升降机械有极片，无真空信号报警
	Mach_Control.Ca_b.Ca_CarryingFalg :=FALSE;
END_IF
		
		
		
		

//负极取片搬运在叠片过程中的真空报警处理
Ca_AlarmTON[15].IN:=NOT arrCyCtrl[arrCyNo.ElectValveName.CaCarryingVacuum2].Io.DIOnSwitch AND Mach_Control.Ca_b.Ca_CarryingFalg 
	 AND  arrAxisCtrl[AxiseNo.AxisName.CaCarryingLine2].Status.Moving AND NOT Mach_Control.U.EmptyRunMode
	AND NOT  arrCyCtrl[arrCyNo.ElectValveName.CaCarryingVacuum2].Io.DOStatus1 AND NOT Bnt_Blueflaging
	AND  arrAxisCtrl[AxiseNo.VirAxisName.VirMain].Status.fActPos>1  AND  arrAxisCtrl[AxiseNo.VirAxisName.VirMain].Status.fActPos<232 ;
	
	IF  Ca_AlarmTON[15].Q THEN  
		CCD.CaRec.Finish.RectifyResult:=0;//拍照结果清零
		Mach_Control.Ca_b.Error[32]:=TRUE;	   //负极取片升降真空叠片过程中真空报警
		Mach_Control.Ca_b.Ca_CarryingFalg :=FALSE;
		arrCyCtrl[arrCyNo.ElectValveName.CaCarryingVacuum2]	.Cmd.bON:=TRUE;//负极搬运2真空破
		arrCyCtrl[arrCyNo.ElectValveName.CaCarryingVacuum2]	.Cmd.bOFF:=FALSE;//负极搬运2真空破
	END_IF
	//搬运平移在叠片过程中报警时，纠偏平台拍照有无片来确定是否掉片到纠偏平台
	IF Mach_Control.Ca_b.Error[32] AND rCa_AlarmReset.Q  THEN
		//CCD.CaRec.Finish.RectifyResult:=0;//拍照结果清零
		Mach_Control.Ca_b.Ca_CCDStart :=TRUE;//启动CCD拍照
		CCD.CaRec.Start.iPhotoDo:=1;//启动CCD第二次拍照
	END_IF
	IF Mach_Control.Ca_b.Error[32] AND (CCD.CaRec.Finish.RectifyResult=3  OR  Mach_Control.U.CCD_ChosesHMI) AND rCa_AlarmReset.Q  THEN
		Mach_Control.Ca_b.Error[32]:=FALSE;
		Mach_Control.Ca_b.Error[33]:=FALSE;//纠偏平台有片，请拿走
	ELSIF Mach_Control.Ca_b.Error[32] AND (CCD.CaRec.Finish.RectifyResult<>3  AND NOT   Mach_Control.U.CCD_ChosesHMI)THEN
		Mach_Control.Ca_b.Error[33]:=TRUE;//纠偏平台有片，请拿走
	END_IF
	
	

	
//负极叠片搬运升降真空信号与有无极片标记信号不一致
Ca_AlarmTON[5].IN:=(arrCyCtrl[arrCyNo.ElectValveName.CaDTCarryingVacuum].Io.DIOnSwitch OR Mach_Control.se.CaDTCarryingJROnSwitch) 
    AND NOT Mach_Control.Ca_b.Ca_DPCarryingFalg 
	AND NOT Mach_Control.U.EmptyRunMode AND Mach_Control.U.DT_iMode=1 AND iEmptyFoldStep[1]=0 AND DP_Step0<1000 AND DP_Step0>3100
	AND NOT  arrCyCtrl[arrCyNo.ElectValveName.CaDTCarryingVacuum].Io.DOStatus1  AND NOT DP_CheseCam  AND NOT Bnt_Blueflaging;//AND NOT Blueflaging
	IF  Ca_AlarmTON[5].Q THEN
		IF  arrCyCtrl[arrCyNo.ElectValveName.CaDTCarryingVacuum].Io.DIOnSwitch THEN
		   Mach_Control.Ca_b.Error[5]:=TRUE;//负极叠台搬运升降有真空信号，无极片报警
		END_IF   
		IF Mach_Control.se.CaDTCarryingJROnSwitch THEN
		   Mach_Control.Ca_b.Error[37]:=TRUE;//负极叠台搬运升降有真空信号，无极耳报警
		END_IF
	END_IF
	
//负极叠台搬运在取片过程中的真空报警处理
Ca_AlarmTON[16].IN:=(NOT arrCyCtrl[arrCyNo.ElectValveName.CaDTCarryingVacuum].Io.DIOnSwitch OR NOT Mach_Control.se.CaDTCarryingJROnSwitch) 
    AND Mach_Control.Ca_b.Ca_DPCarryingFalg AND NOT Mach_Control.U.EmptyRunMode  AND
	arrAxisCtrl[AxiseNo.AxisName.CaDTCarryingUpDown].Status.fActPos<=(arrAxisPar[AxiseNo.AxisName.CaDTCarryingUpDown].arrTargetPoint[2]-5)AND  (Ca_Step2=6666 OR Ca_Step2=0) 
	AND NOT  arrCyCtrl[arrCyNo.ElectValveName.CaDTCarryingVacuum].Io.DOStatus1 AND  arrAxisCtrl[AxiseNo.AxisName.CaDTCarryingLine].Status.NoMoving  AND iEmptyFoldStep[1]=0
	AND (DP_Step0<1000 OR DP_Step0>3100)  ;
	
	IF  Ca_AlarmTON[16].Q THEN
		//CCD.CaRec.Finish.RectifyResult:=0;//拍照结果清零
		IF   NOT arrCyCtrl[arrCyNo.ElectValveName.CaDTCarryingVacuum].Io.DIOnSwitch THEN
	    	Mach_Control.Ca_b.Error[34]:=TRUE;//负极叠台搬运升降有极片，无真空信号反馈
		END_IF		
		IF NOT Mach_Control.se.CaDTCarryingJROnSwitch THEN
		   Mach_Control.Ca_b.Error[39]:=TRUE;//负极叠台搬运升降有极耳无真空报警
		END_IF				
		Mach_Control.Ca_b.Ca_DPCarryingFalg:=FALSE;
		arrCyCtrl[arrCyNo.ElectValveName.CaDTCarryingVacuum].Cmd.bON:=TRUE;//负极叠片搬运升降真空破
		arrCyCtrl[arrCyNo.ElectValveName.CaDTCarryingVacuum].Cmd.bOFF:=FALSE;//负极叠片搬运升降真空破
	END_IF	
	//叠台搬运平移在取片过程中报警时，纠偏平台拍照有无片来确定是否掉片到纠偏平台
	IF (Mach_Control.Ca_b.Error[34] OR Mach_Control.Ca_b.Error[39]) AND rCa_AlarmReset.Q  THEN
		//CCD.CaRec.Finish.RectifyResult:=0;//拍照结果清零
		Mach_Control.Ca_b.Ca_CCDStart :=TRUE;//启动CCD拍照
		CCD.CaRec.Start.iPhotoDo:=1;//启动CCD第二次拍照
	END_IF
	IF (Mach_Control.Ca_b.Error[34]OR Mach_Control.Ca_b.Error[39]) AND (CCD.CaRec.Finish.RectifyResult=3  OR  Mach_Control.U.CCD_ChosesHMI) AND rCa_AlarmReset.Q  THEN
		Mach_Control.Ca_b.Error[34]:=FALSE;//叠台升降取片过程中真空报警，
		Mach_Control.Ca_b.Error[39]:=FALSE;//负极叠台搬运升降有极耳无真空报警
		Mach_Control.Ca_b.Error[33]:=FALSE;//纠偏平台有片，请拿走
	ELSIF (Mach_Control.Ca_b.Error[34] OR Mach_Control.Ca_b.Error[39]) AND (CCD.CaRec.Finish.RectifyResult<>3  AND NOT   Mach_Control.U.CCD_ChosesHMI)THEN
		Mach_Control.Ca_b.Error[33]:=TRUE;//纠偏平台有片，请拿走
	END_IF
	
	
	
//负极叠台搬运在叠片过程中的真空报警处理
Ca_AlarmTON[6].IN:=(NOT arrCyCtrl[arrCyNo.ElectValveName.CaDTCarryingVacuum].Io.DIOnSwitch OR NOT Mach_Control.se.CaDTCarryingJROnSwitch) 
    AND Mach_Control.Ca_b.Ca_DPCarryingFalg 
	AND NOT Mach_Control.U.EmptyRunMode  AND   (Ca_Step2=6666 OR Ca_Step2=0) 
	AND arrAxisCtrl[AxiseNo.VirAxisName.VirMain].Status.fActPos<232 AND NOT Bnt_Blueflaging  AND arrAxisCtrl[AxiseNo.VirAxisName.VirMain].Status.fActPos>1 
	AND NOT  arrCyCtrl[arrCyNo.ElectValveName.CaDTCarryingVacuum].Io.DOStatus1 AND  arrAxisCtrl[AxiseNo.VirAxisName.VirMain].Status.Moving
	AND  arrAxisCtrl[AxiseNo.AxisName.CaDTCarryingLine].Status.Moving  ;
	
	IF  Ca_AlarmTON[6].Q THEN
		//Mach_Control.DT_b.OverhandResult:=0;
		IF   NOT arrCyCtrl[arrCyNo.ElectValveName.CaDTCarryingVacuum].Io.DIOnSwitch THEN
		   Mach_Control.Ca_b.Error[6]:=TRUE;//负极叠台搬运升降有极片，无真空信号反馈
		END_IF	
		IF NOT Mach_Control.se.CaDTCarryingJROnSwitch THEN
		   Mach_Control.Ca_b.Error[38]:=TRUE;//负极叠台搬运升降有极耳无真空报警
		END_IF			
		
		Ca_Number:=TRUE;
		Mach_Control.Ca_b.Ca_DPCarryingFalg:=FALSE;
		arrCyCtrl[arrCyNo.ElectValveName.CaDTCarryingVacuum].Cmd.bON:=TRUE;//负极叠片搬运升降真空破
		arrCyCtrl[arrCyNo.ElectValveName.CaDTCarryingVacuum].Cmd.bOFF:=FALSE;//负极叠片搬运升降真空破
	END_IF	
	//负极叠台搬运升降真空报警，电芯上有片，请拿掉
	Ca_AlarmTON[9].IN:=(Mach_Control.Ca_b.Error[6] OR Mach_Control.Ca_b.Error[38] )  AND Mach_Control.DT_b.OverhandResult<>3 AND NOT Mach_Control.U.CCD_ChosesHMI  ;	
	IF  Ca_AlarmTON[9].Q THEN
		Mach_Control.Ca_b.Error[22]:=TRUE;//负极叠台搬运升降真空报警，电芯上有片，请拿掉
	END_IF
	IF fCa_AlarmRest.Q AND  Mach_Control.Ca_b.Error[22] AND arrAxisCtrl[AxiseNo.VirAxisName.VirMain].Status.fActPos<1 THEN
		CCD.Over.Start.iPhotoDo:=2;
		Mach_Control.DT_b.CDD_OverStart:=TRUE;
	END_IF 
	IF Mach_Control.Ca_b.Error[22] AND Mach_Control.DT_b.OverhandResult=3   AND rCa_AlarmReset.Q  THEN
		Mach_Control.Ca_b.Error[22]:=FALSE;//复位电芯有片报警
		Mach_Control.DT_b.OverhandResult:=0;
	END_IF	
	
	//负极叠台搬运升降真空报警，电芯上无掉片
	Ca_AlarmTON[10].IN:=(Mach_Control.Ca_b.Error[6] OR Mach_Control.Ca_b.Error[38]) AND Mach_Control.DT_b.OverhandResult=3 AND NOT Mach_Control.U.CCD_ChosesHMI    ;	
	IF  Ca_AlarmTON[10].Q THEN
			Mach_Control.Ca_b.Error[23]:=TRUE;//负极叠台搬运升降真空报警，电芯上无掉片
	END_IF	

	


	

		

//负极纠偏平台真空信号与有无料标记不一致报警
Ca_AlarmTON[7].IN:=arrCyCtrl[arrCyNo.ElectValveName.CadeviationVacuum].Io.DIOnSwitch AND NOT Mach_Control.Ca_b.Ca_deviationFalg 
	AND NOT Mach_Control.U.EmptyRunMode AND arrAxisCtrl[AxiseNo.AxisName.CaCarryingUpDown2].Status.Homed  
	AND arrAxisCtrl[AxiseNo.AxisName.CaDTCarryingUpDown].Status.fActPos<=(arrAxisPar[AxiseNo.AxisName.CaDTCarryingUpDown].arrTargetPoint[4]+5) 
	AND iEmptyFoldStep[1]=0 AND (DP_Step0<1000 OR DP_Step0>3100)   ;
		IF  Ca_AlarmTON[7].Q THEN
			Mach_Control.Ca_b.Error[7]:=TRUE;//纠偏平台无片极，有真空信号报警
		END_IF

Ca_AlarmTON[8].IN:=NOT arrCyCtrl[arrCyNo.ElectValveName.CadeviationVacuum].Io.DIOnSwitch AND Mach_Control.Ca_b.Ca_deviationFalg 
	AND NOT Mach_Control.U.EmptyRunMode AND	arrAxisCtrl[AxiseNo.AxisName.CaCarryingUpDown2].Status.Homed  
	AND arrAxisCtrl[AxiseNo.AxisName.CaCarryingUpDown2].Status.fActPos<=(arrAxisPar[AxiseNo.AxisName.CaCarryingUpDown2].arrTargetPoint[4]+5) 
	AND iEmptyFoldStep[1]=0 AND (DP_Step0<1000 OR DP_Step0>3100) AND NOT Mach_Control.Ca_b.Ca_VacuumErrorNG ;	
		IF  Ca_AlarmTON[8].Q THEN
			Mach_Control.Ca_b.Error[8]:=TRUE;//纠偏平台有极片，无真空报警
			Mach_Control.Ca_b.Ca_VacuumErrorNG:=TRUE;//负极抛真空NG料标志			
		END_IF



IF fCa_AlarmRest.Q AND  Mach_Control.Ca_b.Error[24] AND arrAxisCtrl[AxiseNo.VirAxisName.VirMain].Status.fActPos<1 THEN		
	Mach_Control.Ca_b.Ca_CCDStart :=TRUE;//启动CCD拍照
	CCD.CaRec.Start.iPhotoDo:=1;//启动CCD第二次拍照
END_IF
//负极纠偏平台片未排掉报警
IF Mach_Control.Ca_b.Error[24] AND CCD.CaRec.Finish.RectifyResult=3  AND rCa_AlarmReset.Q  THEN
	Mach_Control.Ca_b.Error[24]:=FALSE;
END_IF
//负极纠偏平台连续NG报警
IF Mach_Control.Ca_b.Ca_CCD_amount>=3 AND NOT Mach_Control.Ca_b.Error[21] THEN	
		Mach_Control.Ca_b.Error[21]:=TRUE;//负极纠偏平台连续NG报警
END_IF



//负极取料报警复位
rCa_AlarmReset(CLK:=Sys_Control.btn.System_Rrestbtn , Q=> );//负极报警复位上升沿
fCa_AlarmRest(CLK:=Sys_Control.btn.System_Rrestbtn  , Q=> );//负极报警复位下降沿
IF Mach_Control.U.DT_iMode=3 THEN//在手动状态下，复位报警
	
		IF Mach_Control.Ca_b.Error[2] AND NOT Mach_Control.Ca_b.Ca_SegbeltFalg AND rCa_AlarmReset.Q THEN
				//Mach_Control.Ca_b.Ca_SegbeltFalg:=FALSE;
				//Ca_StandbyStep2:=0;
		END_IF
		
		//IF Mach_Control.Ca_b.Error[4] AND rCa_AlarmReset.Q THEN
			//	Mach_Control.Ca_b.Ca_CarryingFalg:=FALSE;
		//END_IF
		
		IF (Mach_Control.Ca_b.Error[6] OR Mach_Control.Ca_b.Error[38]) AND rCa_AlarmReset.Q THEN
				Mach_Control.Ca_b.Ca_DPCarryingFalg:=FALSE;
		END_IF
//20240105临时屏蔽
	(*		
		IF Mach_Control.Ca_b.Error[8] AND rCa_AlarmReset.Q THEN
				 Mach_Control.Ca_b.Ca_deviationFalg:=FALSE;
		END_IF
	*)	
		IF Mach_Control.Ca_b.Error[21] AND rCa_AlarmReset.Q THEN
				 Mach_Control.Ca_b.Ca_CCD_amount:=0	;	 
		END_IF
		
		
		
																	//20240105临时屏蔽	
		IF ((Mach_Control.Ca_b.Error[4]AND NOT Mach_Control.Ca_b.Ca_CarryingFalg) OR Mach_Control.Ca_b.Error[6] OR Mach_Control.Ca_b.Error[38] ) AND rCa_AlarmReset.Q   THEN
			Ca_StandbyStep0:=0;
			Ca_Step0:=0;
			Ca_Step1:=0;
			Ca_Step2:=0;
			Ca_Step3:=0;
		END_IF
		
		//报警状态复位
		IF fCa_AlarmRest.Q AND NOT Mach_Control.Ca_b.Error[22] AND NOT Mach_Control.Ca_b.Error[4]  AND  NOT Mach_Control.Ca_b.Error[6]   
		AND NOT Mach_Control.Ca_b.Error[32] AND NOT  Mach_Control.Ca_b.Error[24] AND NOT Mach_Control.Ca_b.Error[34] 
        AND NOT  Mach_Control.Ca_b.Error[38] AND NOT  Mach_Control.Ca_b.Error[39]  THEN
			MEMSET(ADR(Mach_Control.Ca_b.Error),0,SIZEOF(Mach_Control.Ca_b.Error)); // 负极取片报警复位	
			//CaOverNGcount:=0;
			arrAxisCtrl[AxiseNo.AxisName.CaDTCarryingLine].Cmd.bStop:=FALSE;
		END_IF
		
		IF CaOverNGcount>=3 AND fCa_AlarmRest.Q  THEN
		   CaOverNGcount:=0;
		END_IF
		
		IF Mach_Control.Ca_b.Ca_DTqr AND Mach_Control.Ca_b.Error[4]   THEN
				Mach_Control.Ca_b.Error[4]:=FALSE;
				Mach_Control.Ca_b.Ca_CarryingFalg:=FALSE;
		END_IF
		
		IF Mach_Control.Ca_b.Ca_DTqr AND  (Mach_Control.Ca_b.Error[6] OR  Mach_Control.Ca_b.Error[38]) THEN
				Mach_Control.Ca_b.Error[6]:=FALSE;
				Mach_Control.Ca_b.Error[38]:=FALSE;
				Mach_Control.Ca_b.Ca_DPCarryingFalg:=FALSE;
		END_IF
		
		IF (Mach_Control.Ca_b.Error[9] OR Ca_RectifydevStep=9999) AND fCa_AlarmRest.Q THEN
				Mach_Control.Ca_b.Error[9]:=FALSE;
				Ca_RectifydevStep:=0;
				CCD.CaRec.Finish.RectifyX1:=0;
				CCD.CaRec.Finish.RectifyX2:=0;
				CCD.CaRec.Finish.RectifyY:=0;		
				CCD.CaRec.Finish.RectifyResult:=0;//拍照结果清零		
		END_IF
		
		IF fCa_AlarmRest.Q THEN		
			IF 9991<=Ca_StandbyStep0 AND  Ca_StandbyStep0<=10000 THEN
				Ca_StandbyStep0:=1000;
				Ca_Step0:=0;
				Ca_Step1:=0;
				Ca_Step2:=0;
				Ca_Step3:=0;
			END_IF
		END_IF
		
END_IF

     Ca_dppy_Xzb:=arrAxisPar[AxiseNo.AxisName.CaCarryingLine2].arrTargetPoint[2]+arrAxisCtrl[AxiseNo.AxisName.CaDTCarryingLine].Status.fActPos;
    IF Ca_Step3=20 AND NOT arrAxis[AxiseNo.AxisName.CaDTCarryingLine].Status.Coupled AND NOT  arrAxis[AxiseNo.AxisName.CaCarryingLine2].Status.Coupled AND arrAxis[AxiseNo.VirAxisName.VirMain].Status.NotMoving  
		  AND arrAxisCtrl[AxiseNo.AxisName.CaCarryingLine2].Status.Homed AND arrAxisCtrl[AxiseNo.AxisName.CaDTCarryingLine].Status.Homed AND NOT arrAxisCtrl[AxiseNo.AxisName.CaCarryingLine2].Cmd.arrbRealPoint[1]
          AND ABS( (arrAxisPar[AxiseNo.AxisName.CaCarryingLine2].arrTargetPoint[2]+arrAxisCtrl[AxiseNo.AxisName.CaDTCarryingLine].Status.fActPos)-arrAxisCtrl[AxiseNo.AxisName.CaCarryingLine2].Status.fActPos)
            <(ABS(arrAxisPar[AxiseNo.AxisName.CaCarryingLine2].arrTargetPoint[2]-arrAxisPar[AxiseNo.AxisName.CaCarryingLine2].arrTargetPoint[1])+arrAxisPar[AxiseNo.AxisName.CaDTCarryingLine].arrTargetPoint[1]-20) THEN
			Mach_Control.Ca_b.Error[26]:=TRUE;//负极搬运平移防撞软限位报警
	END_IF
	
	CaError_r(CLK:=  Mach_Control.Ca_b.Error[26] , Q=> );
	IF CaError_r.Q THEN 
		   arrAxisCtrl[AxiseNo.AxisName.CaCarryingLine2].Cmd.bStop:=TRUE;
		   arrAxisCtrl[AxiseNo.AxisName.CaDTCarryingLine].Cmd.bStop :=TRUE;	
	END_IF
	
    IF  P2M2_sysControl.btn.System_Rrestbtn  THEN
      	 arrAxisCtrl[AxiseNo.AxisName.CaCarryingLine2].Cmd.bStop:=FALSE;
     	  arrAxisCtrl[AxiseNo.AxisName.CaDTCarryingLine].Cmd.bStop :=FALSE;
	END_IF

IF Mach_Control.U.DT_iMode=3 THEN//在手动状态下，复位报警	
		IF Mach_Control.Ca_b.Error[28] AND DP_Step0=3070 AND rCa_AlarmReset.Q THEN
				Mach_Control.Ca_b.Ca_DPCarryingFalg:=FALSE;
		END_IF
END_IF

//ccdJ拍照检测返回结果超时报警
rCaCCDStart(CLK:=Mach_Control.Ca_b.Ca_CCDStart, Q=> );
IF rAnCCDStart.Q THEN
	 CaCCDMark:=TRUE;
END_IF
 
IF CaCCDMark AND CCD. CaRec.Finish.RectifyResult=0 AND NOT Mach_Control.U.CCD_ChosesHMI THEN
		IF NOT  Ca_AlarmTon[12].Q THEN
			 	Ca_AlarmTon[12].IN:=TRUE;
		ELSE	
				Mach_Control.Ca_b.Error[18] :=TRUE;//负极CCD纠偏平台检测返回结果超时
				CaCCDMark :=FALSE;
		END_IF
ELSE
		 Ca_AlarmTon[12].IN:=FALSE;
END_IF

IF (Mach_Control.Ca_b.Error[18] AND Sys_Control.btn.System_Rrestbtn) OR
    (CCD. CaRec.Finish.RectifyResult<>0 AND  CaCCDMark AND  Ca_AlarmTon[13].Q ) THEN
	   CaCCDMark :=FALSE;
	   Ca_AlarmTon[12].IN:=FALSE;
END_IF	

IF Mach_Control.U.DT_iMode=1 AND  rCaUse[4].Q THEN
 Par.stDT_date.Ca_sucker1_JS :=Par.stDT_date.Ca_sucker1_JS+1;
END_IF

IF( HMI_Hour>=7  AND HMI_Hour<9) OR (HMI_Hour>=19  AND HMI_Hour<21) THEN
      IF Par.stDT_date.Ca_sucker1_JS>=Par.stDT_date.Ca_sucker1Set THEN
	      Mach_Control.Ca_b.Error[43]:=TRUE;//负极送片搬运吸盘计数到达设定值
      END_IF
END_IF
IF Mach_Control.DT_b.Ca_sucker1_JSclear THEN
   Par.stDT_date.Ca_sucker1_JS:=0;
END_IF  

IF Mach_Control.U.DT_iMode=1 AND  rCaUse[5].Q THEN
 Par.stDT_date.Ca_sucker2_JS :=Par.stDT_date.Ca_sucker2_JS+1;
END_IF

IF( HMI_Hour>=7  AND HMI_Hour<9) OR (HMI_Hour>=19  AND HMI_Hour<21) THEN
      IF Par.stDT_date.Ca_sucker2_JS>=Par.stDT_date.Ca_sucker2Set THEN
	      Mach_Control.Ca_b.Error[44]:=TRUE;//负极叠台搬运吸盘计数到达设定值
      END_IF
END_IF
IF Mach_Control.DT_b.Ca_sucker2_JSclear THEN
   Par.stDT_date.Ca_sucker2_JS:=0;
END_IF  
IF Mach_Control.U.DT_iMode=1 AND  rCaUse[6].Q THEN
 Par.stDT_date.Ca_sucker3_JS :=Par.stDT_date.Ca_sucker3_JS+1;
END_IF

IF( HMI_Hour>=7  AND HMI_Hour<9) OR (HMI_Hour>=19  AND HMI_Hour<21) THEN
      IF Par.stDT_date.Ca_sucker3_JS>=Par.stDT_date.Ca_sucker3Set THEN
	      Mach_Control.Ca_b.Error[45]:=TRUE;//负极流水线搬运吸盘计数到达设定值
      END_IF
END_IF
IF Mach_Control.DT_b.Ca_sucker3_JSclear THEN
   Par.stDT_date.Ca_sucker3_JS:=0;
END_IF  
(*
IF Ca_CCDNG>=10 THEN
		Mach_Control.Ca_b.Error[12]:=TRUE;//负极NG收纳盒满料报警
END_IF

IF Mach_Control.Ca_b.Error[12] AND P2M2_sysControl.btn.System_Rrestbtn THEN
		 Mach_Control.Ca_b.Error[12]:=FALSE;
		 Ca_CCDNG:=0;
END_IF

*)
END_ACTION

ACTION Ca_Cahebelt:
Ca_TON[9].IN:=Mach_Control.Ca_b.bCa_PoleHave;
IF Ca_TON[9].Q THEN
	Mach_Control.Ca_b.bCa_PoleHave:=FALSE;//负极取流水线极片完成，
END_IF


//取料中信号复位
Ca_TON[10].IN:= NOT  arrAxisCtrl[AxiseNo.AxisName.CaCarryingUpDown1].Cmd.arrbRealPoint[1] AND Mach_Control.Ca_b.JumpPiceReady AND Mach_Control.Ca_b.Ca_MainBelting;
IF Ca_TON[10].Q THEN
	IF NOT  arrAxisCtrl[AxiseNo.AxisName.CaCarryingUpDown1].Cmd.arrbRealPoint[1] THEN		
		arrAxisCtrl[AxiseNo.AxisName.CaCarryingUpDown1].Cmd.iGoSetPos:=1;//负极送片搬运升降上升至初始高度	
	ELSE
		arrAxisCtrl[AxiseNo.AxisName.CaCarryingUpDown1].Cmd.iGoSetPos:=0;//负极送片搬运升降上升至初始高度	
	END_IF
END_IF
Ca_TON[11].IN:=arrAxisCtrl[AxiseNo.AxisName.CaCarryingUpDown1].Cmd.arrbRealPoint[1] AND Mach_Control.Ca_b.JumpPiceReady AND Mach_Control.Ca_b.Ca_MainBelting;
IF Ca_TON[11].Q  THEN
	Ca_StandbyStep2:=0;
	Mach_Control.Ca_b.Ca_BeltDone:=TRUE;//取流水线取极片完成
	Mach_Control.Ca_b.Ca_MainBelting:=FALSE;//正极搬运升降取极片中
END_IF




IF Mach_Control.U.DT_iMode=1 OR AG  THEN//在自动状态下
//负极模切分段皮带极片自动
CASE Ca_StandbyStep2  OF
0://判断取模切分板皮带机械手有无料标记
	IF NOT DP_SinStepe THEN
		IF   arrAxisCtrl[AxiseNo.AxisName.CaCarryingUpDown1].Status.Enabled  AND  arrAxisCtrl[AxiseNo.AxisName.CaCarryingLine1].Status.Enabled 
		AND  arrAxisCtrl[AxiseNo.AxisName.CaCarryingWhirling1].Status.Enabled  THEN
			IF Mach_Control.Ca_b.Ca_SegbeltFalg  THEN//负极取模切分段机械手有极片标记
				DT_SingeMode();//单步选择
				Ca_StandbyStep2:=100;
			ELSE//负极取模切分段机械手无料
				
				DT_SingeMode();//单步选择
				Ca_StandbyStep2:=10;
			END_IF
		END_IF
	END_IF
10://负极送片搬运升降轴上升至安全位，真空关闭
	IF NOT DP_SinStepe THEN
		arrCyCtrl[arrCyNo.ElectValveName.CaCarryingVacuum1]	.Cmd.bOFF:=TRUE;//负极搬运1真空关
		arrCyCtrl[arrCyNo.ElectValveName.CaCarryingVacuum1]	.Cmd.bON:=FALSE;//负极搬运1真空开
		IF arrAxisCtrl[AxiseNo.AxisName.CaCarryingUpDown1].Status.Homed AND arrAxisCtrl[AxiseNo.AxisName.CaCarryingUpDown1].Status.NoMoving AND 
			NOT arrAxisCtrl[AxiseNo.AxisName.CaCarryingUpDown1].Status.Error THEN
				IF arrAxisCtrl[AxiseNo.AxisName.CaCarryingUpDown1].Cmd.arrbRealPoint[1] THEN
					arrAxisCtrl[AxiseNo.AxisName.CaCarryingUpDown1].Cmd.iGoSetPos:=0;
					DT_SingeMode();//单步选择
					Ca_StandbyStep2:=20;
				ELSE
					arrAxisCtrl[AxiseNo.AxisName.CaCarryingUpDown1].Cmd.iGoSetPos:=1;//负极搬运升降1移动至初始高度
				END_IF
		END_IF
	END_IF
20://负极送片搬运平移至模切分段皮带取料位,负极搬运旋转1旋转至初始位
	IF NOT DP_SinStepe THEN
		IF arrAxisCtrl[AxiseNo.AxisName.CaCarryingUpDown1].Cmd.arrbRealPoint[1] AND  arrAxisCtrl[AxiseNo.AxisName.CaCarryingLine1].Status.Homed AND 
			arrAxisCtrl[AxiseNo.AxisName.CaCarryingLine1].Status.NoMoving AND NOT arrAxisCtrl[AxiseNo.AxisName.CaCarryingLine1].Status.Error THEN
			IF arrAxisCtrl[AxiseNo.AxisName.CaCarryingLine1].Cmd.arrbRealPoint[1] THEN
				arrAxisCtrl[AxiseNo.AxisName.CaCarryingLine1].Cmd.iGoSetPos:=0;
			ELSE
				arrAxisCtrl[AxiseNo.AxisName.CaCarryingLine1].Cmd.iGoSetPos:=1;//负极搬运升降1移动至初始高度
			END_IF
		END_IF
		IF arrAxisCtrl[AxiseNo.AxisName.CaCarryingUpDown1].Cmd.arrbRealPoint[1] AND  arrAxisCtrl[AxiseNo.AxisName.CaCarryingWhirling1].Status.Homed AND
			 arrAxisCtrl[AxiseNo.AxisName.CaCarryingWhirling1].Status.NoMoving AND NOT arrAxisCtrl[AxiseNo.AxisName.CaCarryingWhirling1].Status.Error THEN
			IF arrAxisCtrl[AxiseNo.AxisName.CaCarryingWhirling1].Cmd.arrbRealPoint[1] THEN
				arrAxisCtrl[AxiseNo.AxisName.CaCarryingWhirling1].Cmd.iGoSetPos:=0;
			ELSE
				arrAxisCtrl[AxiseNo.AxisName.CaCarryingWhirling1].Cmd.iGoSetPos:=1;//负极搬运旋转至初始位
			END_IF
		END_IF
		IF arrAxisCtrl[AxiseNo.AxisName.CaCarryingLine1].Cmd.arrbRealPoint[1]  AND arrAxisCtrl[AxiseNo.AxisName.CaCarryingWhirling1].Cmd.arrbRealPoint[1] THEN
			DT_SingeMode();//单步选择
			Ca_StandbyStep2:=30;
		END_IF
	END_IF

	

100://负极送片搬运升降轴上升至安全位，真空关闭
	IF NOT DP_SinStepe THEN
		IF arrAxisCtrl[AxiseNo.AxisName.CaCarryingUpDown1].Status.Homed AND arrAxisCtrl[AxiseNo.AxisName.CaCarryingUpDown1].Status.NoMoving AND 
			NOT arrAxisCtrl[AxiseNo.AxisName.CaCarryingUpDown1].Status.Error THEN
			IF arrAxisCtrl[AxiseNo.AxisName.CaCarryingUpDown1].Cmd.arrbRealPoint[1] THEN
						arrAxisCtrl[AxiseNo.AxisName.CaCarryingUpDown1].Cmd.iGoSetPos:=0;
						DT_SingeMode();//单步选择
						Ca_StandbyStep2:=110;
			ELSE
				arrAxisCtrl[AxiseNo.AxisName.CaCarryingUpDown1].Cmd.iGoSetPos:=1;//负极搬运升降1移动至初始高度
			END_IF
		END_IF
	END_IF
110://负极送片搬运平移至模切分段皮带放极片位, 负极搬运旋转1旋转至放位
	IF NOT DP_SinStepe THEN
		IF arrAxisCtrl[AxiseNo.AxisName.CaCarryingUpDown1].Cmd.arrbRealPoint[1] AND  arrAxisCtrl[AxiseNo.AxisName.CaCarryingLine1].Status.Homed AND 
			arrAxisCtrl[AxiseNo.AxisName.CaCarryingLine1].Status.NoMoving AND NOT arrAxisCtrl[AxiseNo.AxisName.CaCarryingLine1].Status.Error THEN
			IF arrAxisCtrl[AxiseNo.AxisName.CaCarryingLine1].Cmd.arrbRealPoint[2] THEN
				arrAxisCtrl[AxiseNo.AxisName.CaCarryingLine1].Cmd.iGoSetPos:=0;
			ELSE
				arrAxisCtrl[AxiseNo.AxisName.CaCarryingLine1].Cmd.iGoSetPos:=2;//负极搬运升降1移动至放极片位
			END_IF
		END_IF
		IF arrAxisCtrl[AxiseNo.AxisName.CaCarryingUpDown1].Cmd.arrbRealPoint[1] AND  arrAxisCtrl[AxiseNo.AxisName.CaCarryingWhirling1].Status.Homed AND
			 arrAxisCtrl[AxiseNo.AxisName.CaCarryingWhirling1].Status.NoMoving AND NOT arrAxisCtrl[AxiseNo.AxisName.CaCarryingWhirling1].Status.Error THEN
			IF arrAxisCtrl[AxiseNo.AxisName.CaCarryingWhirling1].Cmd.arrbRealPoint[2] THEN
				arrAxisCtrl[AxiseNo.AxisName.CaCarryingWhirling1].Cmd.iGoSetPos:=0;
			ELSE
				arrAxisCtrl[AxiseNo.AxisName.CaCarryingWhirling1].Cmd.iGoSetPos:=2;//负极搬运旋转至放极片位
			END_IF
		END_IF
		IF arrAxisCtrl[AxiseNo.AxisName.CaCarryingLine1].Cmd.arrbRealPoint[2]  AND arrAxisCtrl[AxiseNo.AxisName.CaCarryingWhirling1].Cmd.arrbRealPoint[2] THEN
			DT_SingeMode();//叠片单步选择
			Ca_StandbyStep2:=120;
		END_IF
	END_IF
120://判断负极流水线是否允许放极片  OR Mach_Control.U.EmptyRunMode
	IF NOT DP_SinStepe THEN
		IF Mach_Control.Ca_b.Ca_CacheBeltFLOK AND  Mach_Control.Ca_b.Ca_SegbeltFalg THEN
			DT_SingeMode();//单步选择
			Ca_StandbyStep2:=130;
		ELSIF NOT Mach_Control.Ca_b.Ca_SegbeltFalg THEN
			Ca_StandbyStep2:=0;
		END_IF
	END_IF
130://负极搬运升降1下降至放极片位
	IF NOT DP_SinStepe THEN
		IF arrAxisCtrl[AxiseNo.AxisName.CaCarryingLine1].Cmd.arrbRealPoint[2]  AND arrAxisCtrl[AxiseNo.AxisName.CaCarryingWhirling1].Cmd.arrbRealPoint[2] AND 
			arrAxisCtrl[AxiseNo.AxisName.CaCarryingUpDown1].Status.Homed AND arrAxisCtrl[AxiseNo.AxisName.CaCarryingUpDown1].Status.NoMoving AND 
			NOT arrAxisCtrl[AxiseNo.AxisName.CaCarryingUpDown1].Status.Error THEN
			IF arrAxisCtrl[AxiseNo.AxisName.CaCarryingUpDown1].Cmd.arrbRealPoint[3] THEN
				arrAxisCtrl[AxiseNo.AxisName.CaCarryingUpDown1].Cmd.iGoSetPos:=0;
				arrCyCtrl[arrCyNo.ElectValveName.CaCarryingVacuum1].Cmd.bOFF:=TRUE;//负极搬运1升降真空关
				arrCyCtrl[arrCyNo.ElectValveName.CaCarryingVacuum1].Cmd.bON:=FALSE;//负极搬运1升降真空关
				arrCyCtrl[arrCyNo.ElectValveName.CaCarryingVacuumBark1].Cmd.bON:=TRUE;//负极搬运1升降破真空开
				arrCyCtrl[arrCyNo.ElectValveName.CaCarryingVacuumBark1].Cmd.bOFF:=FALSE;//负极搬运1升降破真空开
				Mach_Control.Ca_b.Ca_SegbeltFalg:=FALSE;//置位负极取模切分段机械手有极片标记
				Par.stDT_date.Ca_betlCount.0:=TRUE;//置位负极片流水线放片位有片
				Par.stDT_date.Ca_MQ_Slice[1]:=Par.stDT_date.Ca_MQ_Slice[0];
				DT_SingeMode();//单步选择
				Ca_StandbyStep2:=140;
			ELSE
				arrAxisCtrl[AxiseNo.AxisName.CaCarryingUpDown1].Cmd.iGoSetPos:=3;//负极搬运升降1移动至放极片高度
			END_IF
		ELSE
			IF arrAxisCtrl[AxiseNo.AxisName.CaCarryingLine1].Cmd.arrbRealPoint[2] THEN
				arrAxisCtrl[AxiseNo.AxisName.CaCarryingLine1].Cmd.iGoSetPos:=0;
			ELSE
				arrAxisCtrl[AxiseNo.AxisName.CaCarryingLine1].Cmd.iGoSetPos:=2;//负极搬运升降1移动至放极片位
			END_IF	
			IF arrAxisCtrl[AxiseNo.AxisName.CaCarryingWhirling1].Cmd.arrbRealPoint[2] THEN
				arrAxisCtrl[AxiseNo.AxisName.CaCarryingWhirling1].Cmd.iGoSetPos:=0;
			ELSE
				arrAxisCtrl[AxiseNo.AxisName.CaCarryingWhirling1].Cmd.iGoSetPos:=2;//负极搬运旋转至放极片位
			END_IF			
		END_IF
	END_IF
140://负极送片搬运升降轴上升至安全位，真空关闭
	IF NOT DP_SinStepe THEN
		IF arrAxisCtrl[AxiseNo.AxisName.CaCarryingUpDown1].Status.Homed AND arrAxisCtrl[AxiseNo.AxisName.CaCarryingUpDown1].Status.NoMoving AND 
			NOT arrAxisCtrl[AxiseNo.AxisName.CaCarryingUpDown1].Status.Error THEN
			IF arrAxisCtrl[AxiseNo.AxisName.CaCarryingUpDown1].Cmd.arrbRealPoint[1] THEN
				arrAxisCtrl[AxiseNo.AxisName.CaCarryingUpDown1].Cmd.iGoSetPos:=0;
				DT_SingeMode();//单步选择
				Ca_StandbyStep2:=0;
			ELSE
				arrAxisCtrl[AxiseNo.AxisName.CaCarryingUpDown1].Cmd.iGoSetPos:=1;//负极搬运升降1移动至初始高度
			END_IF
		END_IF
	END_IF				
END_CASE	
END_IF


//负极缓存流水线缓存极片自动	
CASE Ca_StandbyStep4 OF
0://判断是否可以补极片,负极搬运升降1轴在安全位，负极搬运各项降2轴在安全位，负极流水线放极片端有极片，负极片流水线取级片端没极片 
	IF NOT Par.stDT_date.Ca_betlCount.5 AND Par.stDT_date.Ca_betlCount.0 AND  Mach_Control.Ca_b.Ca_betlMoveOK  THEN
		IF NOT Mach_Control.se.Offloadingsensor THEN
				Par.stDT_date.Ca_betlCount.4:=FALSE;
		END_IF
		Ca_StandbyStep4:=10;
	ELSIF	Ca_StandbyStep2=120 AND NOT Par.stDT_date.Ca_betlCount.5 AND Par.stDT_date.Ca_betlCount.0  AND  NOT  arrAxisCtrl[AxiseNo.AxisName.CaCarryingUpDown1].Cmd.arrbRealPoint[1] THEN
               // ( arrAxisCtrl[AxiseNo.AxisName.CaCarryingUpDown1].Status.fSetPos > arrAxisPar[AxiseNo.AxisName.CaCarryingUpDown1].arrTargetPoint[1]+0.5 OR
                //  arrAxisCtrl[AxiseNo.AxisName.CaCarryingUpDown1].Status.fSetPos < arrAxisPar[AxiseNo.AxisName.CaCarryingUpDown1].arrTargetPoint[1]-0.5)THEN
		         Mach_Control.Ca_b.Error[41]:=TRUE;//负极缓存皮带准备运动时，负极升降1不在安全位报警	
	END_IF
10://负极流水线皮带向前移动固定距离
	arrAxisCtrl[AxiseNo.AxisName.CaBelt].Cmd.bDynamitcsParSel:=1;	
	arrAxisPar[AxiseNo.AxisName.CaBelt].fTagatTime:=Par.stDT_date.BeltPoistTime;
	arrAxisCtrl[AxiseNo.AxisName.CaBelt].Cmd.fPosition_of_Rel:=Par.stDT_date.BeltPoistSet;
	arrAxisCtrl[AxiseNo.AxisName.CaBelt].Cmd.bMoveRel:=TRUE;	
	Ca_StandbyStep4:=20;
20:
	IF NOT arrAxisCtrl[AxiseNo.AxisName.CaBelt].Cmd.bMoveRel THEN
		Par.stDT_date.Ca_betlCount:=SHL(Par.stDT_date.Ca_betlCount,1);//极片向前移一位
		Ca_StandbyStep4:=31;
	END_IF

31:	
	Par.stDT_date.Ca_MQ_Slice[6]:=Par.stDT_date.Ca_MQ_Slice[5];
	Ca_StandbyStep4:=32;

32:
	Par.stDT_date.Ca_MQ_Slice[5]:=Par.stDT_date.Ca_MQ_Slice[4];
	Ca_StandbyStep4:=33;

33:
	Par.stDT_date.Ca_MQ_Slice[4]:=Par.stDT_date.Ca_MQ_Slice[3];
	Ca_StandbyStep4:=34;

34:	
	Par.stDT_date.Ca_MQ_Slice[3]:=Par.stDT_date.Ca_MQ_Slice[2];
	Ca_StandbyStep4:=35;

35:
	Par.stDT_date.Ca_MQ_Slice[2]:=Par.stDT_date.Ca_MQ_Slice[1];
	Ca_StandbyStep4:=36;

36://复位负极片流水线放片位有片
	MEMSET(ADR(Par.stDT_date.Ca_MQ_Slice[1]),0,SIZEOF(Par.stDT_date.Ca_MQ_Slice[1]));
	Par.stDT_date.Ca_betlCount.0:=FALSE;
	Ca_StandbyStep4:=0;
END_CASE


CASE Ca_StandbyStep2  OF
30://判断模切分段皮带是否允许取极片 OR Mach_Control.U.EmptyRunMode 
	IF NOT DP_SinStepe THEN
		IF Mach_Control.Ca_b.Ca_MainBeltOK THEN
			Mach_Control.Ca_b.Ca_MainBelting:=TRUE;//负极模切分段皮带取极片中
			arrCyCtrl[arrCyNo.ElectValveName.CaCarryingVacuum1]	.Cmd.bON:=TRUE;//负极搬运1真空打开
			arrCyCtrl[arrCyNo.ElectValveName.CaCarryingVacuum1]	.Cmd.bOFF:=FALSE;//负极搬运1真空关闭
			DT_SingeMode();//单步选择
			Ca_StandbyStep2:=35;
		//ELSE
		//	Ca_StandbyStep2:=0;
		END_IF
	END_IF
35://负极搬动升降1下降取极片
	IF NOT DP_SinStepe THEN
		IF arrAxisCtrl[AxiseNo.AxisName.CaCarryingLine1].Cmd.arrbRealPoint[1]  AND arrAxisCtrl[AxiseNo.AxisName.CaCarryingWhirling1].Cmd.arrbRealPoint[1] AND 
			arrAxisCtrl[AxiseNo.AxisName.CaCarryingUpDown1].Status.Homed AND  NOT arrAxisCtrl[AxiseNo.AxisName.CaCarryingUpDown1].Status.Error THEN
			IF arrAxisCtrl[AxiseNo.AxisName.CaCarryingUpDown1].Cmd.arrbRealPoint[2] OR arrAxisCtrl[AxiseNo.AxisName.CaCarryingUpDown1].Status.Moving THEN
				arrAxisCtrl[AxiseNo.AxisName.CaCarryingUpDown1].Cmd.iGoSetPos:=0;
				DT_SingeMode();//单步选择
				Ca_TON[6].IN:=FALSE;
				Ca_StandbyStep2:=40;
			ELSE
				arrAxisCtrl[AxiseNo.AxisName.CaCarryingUpDown1].Cmd.iGoSetPos:=2;//负极搬运升降1移动至初始高度
			END_IF					
		END_IF
	END_IF
40://负极搬动升降1下降取极片
	IF arrAxisCtrl[AxiseNo.AxisName.CaCarryingLine1].Cmd.arrbRealPoint[1]  AND arrAxisCtrl[AxiseNo.AxisName.CaCarryingWhirling1].Cmd.arrbRealPoint[1] AND 
	arrAxisCtrl[AxiseNo.AxisName.CaCarryingUpDown1].Status.Homed AND arrAxisCtrl[AxiseNo.AxisName.CaCarryingUpDown1].Status.NoMoving AND 
	NOT arrAxisCtrl[AxiseNo.AxisName.CaCarryingUpDown1].Status.Error THEN
		IF arrAxisCtrl[AxiseNo.AxisName.CaCarryingUpDown1].Cmd.arrbRealPoint[2] THEN			
			IF NOT Ca_TON[6].Q THEN
				Ca_TON[6].IN:=TRUE;
			ELSE
				//Mach_Control.Ca_b.bCa_PoleHave:=TRUE;//负极取流水线极片完成，复位取片位置极片有无信号
				arrAxisCtrl[AxiseNo.AxisName.CaCarryingUpDown1].Cmd.iGoSetPos:=0;
				//arrCyCtrl[arrCyNo.ElectValveName.CaMQBeltVacuum].Cmd.bOFF:=TRUE;//负极模切分段皮带真空关闭
				//arrCyCtrl[arrCyNo.ElectValveName.CaMQBeltVacuum].Cmd.bON:=FALSE;//负极模切分段皮带真空关闭
				//arrCyCtrl[arrCyNo.ElectValveName.CaMQBeltVacuumBark].Cmd.bON:=TRUE;//负极模切分段皮带破真空打开
				Mach_Control.Ca_b.Ca_SegbeltFalg:=TRUE;//置位负极取模切分段机械手有极片标记
				Par.stDT_date.Ca_MQ_Slice[0]:=Par.stDT_date.CaMQ_MES;//转移皮带上的数据
				DT_SingeMode();//单步选择
				Ca_TON[6].IN:=FALSE;
				Ca_StandbyStep2:=50;								
			END_IF								
		ELSE
			arrAxisCtrl[AxiseNo.AxisName.CaCarryingUpDown1].Cmd.iGoSetPos:=2;//负极搬运升降1移动至初始高度
		END_IF					
	END_IF

50://
	//20240414 wcz
    IF   arrAxisCtrl[AxiseNo.AxisName.CaCarryingUpDown1].Status.fActPos<=(arrAxisPar[AxiseNo.AxisName.CaCarryingUpDown1].arrTargetPoint[2]-3) AND
		 arrAxisCtrl[AxiseNo.AxisName.CaCarryingUpDown1].Status.Moving THEN
			Mach_Control.Ca_b.Ca_MainBelting:=FALSE;//负极模切分段皮带取极片中
			Mach_Control.Ca_b.Ca_BeltDone:=TRUE;//负极取主流水线极片完成		 
			Mach_Control.Ca_b.bCa_PoleHave:=TRUE;//负极取流水线极片完成，复位取片位置极片有无信号
	END_IF

	IF arrAxisCtrl[AxiseNo.AxisName.CaCarryingUpDown1].Status.Homed AND arrAxisCtrl[AxiseNo.AxisName.CaCarryingUpDown1].Status.NoMoving AND 
	NOT arrAxisCtrl[AxiseNo.AxisName.CaCarryingUpDown1].Status.Error THEN
		IF arrAxisCtrl[AxiseNo.AxisName.CaCarryingUpDown1].Cmd.arrbRealPoint[1] THEN
			arrAxisCtrl[AxiseNo.AxisName.CaCarryingUpDown1].Cmd.iGoSetPos:=0;
			Mach_Control.Ca_b.Ca_MainBelting:=FALSE;//负极模切分段皮带取极片中
			Mach_Control.Ca_b.Ca_BeltDone:=TRUE;//负极取主流水线极片完成
			DT_SingeMode();//单步选择
			Ca_StandbyStep2:=0;
		ELSE
			arrAxisCtrl[AxiseNo.AxisName.CaCarryingUpDown1].Cmd.iGoSetPos:=1;//负极搬运升降1移动至初始高度
		END_IF
	END_IF
END_CASE
END_ACTION

ACTION Ca_Cam:
Ca_Cam_ton[1](PT:=T#100MS);
Ca_Cam_ton[2](PT:=T#100MS);
Ca_Cam_ton[3](PT:=T#100MS);
Ca_Cam_ton[4](PT:=T#100MS);
Ca_Cam_ton[5](PT:=T#100MS);
(***********************************负极凸轮表创建************************************************)
(*
      fbCaCrectCamCarryingLine1              :FB_CrectCamMove ;
      fbCaCrectCamCarryingUpDown1       :FB_CrectCamUpDown ;
      fbCaCrectCamCarryingLine2             :FB_CrectCamMove ;
      fbCaCrectCamCarryingUpDown2       :FB_CrectCamUpDown ;
      fbCaCrectCamDTCarryingLine            :FB_CrectCamMove ;
      fbCaCrectCamDTCarryingUpDown     :FB_CrectCamUpDown ;
*)
//负极取流水线搬运平移凸轮创建
fbCaCrectCamCarryingLine1(
	bCreatTable:=                fbCaCrectCamCarryingLine1.bCreatTable , 
	Reset:=                          stSysState.bReset  ,  
	iTable:=                       TableNo.M_CaCarryingLine1  , 
	fMoveLength:=             390 , 
	fMasterKeyPos:=          224 , 
	
	axisMaster:=                 arrAxis[AxiseNo.VirAxisName.CaCarryingVirGM] ,  
    axisSlave:=                    arrAxis[AxiseNo.AxisName.CaCarryingLine1] ,  
	bCreatTableDone=> , 
	bCreatTableError=> , 
	bError=> );

fbCaCrectCamCarryingLine1.bCreatTableDone;
fbCaCrectCamCarryingLine1.bCreatTableError;
fbCaCrectCamCarryingLine1.bError;

//负极取流水线搬运放片升降凸轮创建
fbCaCrectCamCarryingUpDown1(
	bCreatTable:=                         fbCaCrectCamCarryingUpDown1.bCreatTable , 
	Reset:=                                  stSysState.bReset  ,  
	iTable:=                                   TableNo.M_CaCarryingUpDown1   , 
	fMoveLength:=                        18   , //升降轴放片或取片位
	fSaveLength:=                          3, //升降轴安全位
	fInitLength:=						      13,//升降轴耦合初始位
	fMasterKeyPos1:= , //208
	fMasterKeyPos2:= , //256
	fMasterKeyPos3:= , //328

    axisMaster:=                        arrAxis[AxiseNo.VirAxisName.CaCarryingVirGM] ,   
	axisSlave:=                           arrAxis[AxiseNo.AxisName.CaCarryingUpDown1] ,  

	bCreatTableDone=> , 
	bCreatTableError=> , 
	bError=> );
fbCaCrectCamCarryingUpDown1.bCreatTableDone;
fbCaCrectCamCarryingUpDown1.bCreatTableError;
fbCaCrectCamCarryingUpDown1.bError;

//负极取流水线搬运取片升降凸轮创建
fbCaCrectCamCarryingUpDown1_1(
	bCreatTable:=                         fbCaCrectCamCarryingUpDown1_1.bCreatTable , 
	Reset:=                                  stSysState.bReset  ,  
	iTable:=                                   TableNo.M_CaCarryingUpDown1_1   , 
	fMoveLength:=                        18   , //升降轴放片或取片位
	fSaveLength:=                          3, //升降轴安全位
	fInitLength:=						      13,//升降轴耦合初始位
	fMasterKeyPos1:= , //208
	fMasterKeyPos2:= , //256
	fMasterKeyPos3:= , //328

    axisMaster:=                        arrAxis[AxiseNo.VirAxisName.CaCarryingVirGM] ,   
	axisSlave:=                           arrAxis[AxiseNo.AxisName.CaCarryingUpDown1] ,  

	bCreatTableDone=> , 
	bCreatTableError=> , 
	bError=> );
fbCaCrectCamCarryingUpDown1_1.bCreatTableDone;
fbCaCrectCamCarryingUpDown1_1.bCreatTableError;
fbCaCrectCamCarryingUpDown1_1.bError;

//负极取流水线旋转凸轮创建 
fbCaCrectCamCarryingWhirling(
	bCreatTable:=                fbCaCrectCamCarryingWhirling.bCreatTable , 
	Reset:=                          stSysState.bReset  ,  
	iTable:=                       TableNo.M_CaCarryingWhirling1  , 
	fMoveLength:=             390 , 
	fMasterKeyPos:=          170 , //224
	
	axisMaster:=                 arrAxis[AxiseNo.VirAxisName.CaCarryingVirGM] ,  
    axisSlave:=                    arrAxis[AxiseNo.AxisName.CaCarryingWhirling1] ,  
	bCreatTableDone=> , 
	bCreatTableError=> , 
	bError=> );

fbCaCrectCamCarryingWhirling.bCreatTableDone;
fbCaCrectCamCarryingWhirling.bCreatTableError;
fbCaCrectCamCarryingWhirling.bError;




//负极送纠偏平台搬运平移凸轮创建
fbCaCrectCamCarryingLine2.fMoveLength:=ABS(arrAxisPar[AxiseNo.AxisName.CaCarryingLine2].arrTargetPoint[1]-arrAxisPar[AxiseNo.AxisName.CaCarryingLine2].arrTargetPoint[2]);
fbCaCrectCamCarryingLine2(
	bCreatTable:=                fbCaCrectCamCarryingLine2.bCreatTable , 
	Reset:=                          stSysState.bReset  ,  
	iTable:=                       TableNo.M_CaCarryingLine2  , 
	fMoveLength:=             , 
	fMasterKeyPos:=          250 , //
	
	axisMaster:=                 arrAxis[AxiseNo.VirAxisName.VirMain] ,  
    axisSlave:=                    arrAxis[AxiseNo.AxisName.CaCarryingLine2] ,  
	bCreatTableDone=> , 
	bCreatTableError=> , 
	bError=> );

fbCaCrectCamCarryingLine2.bCreatTableDone;
fbCaCrectCamCarryingLine2.bCreatTableError;
fbCaCrectCamCarryingLine2.bError;


(**********20240528SJ***************)
arrAxisPar[AxiseNo.AxisName.CaCarryingUpDown2].arrTargetPoint[10]:=10; //等待高度  参数可调
arrAxisPar[AxiseNo.AxisName.CaCarryingUpDown2].arrTargetPoint[11]:=25; //安全高度  参数可调
arrAxisPar[AxiseNo.AxisName.CaCarryingUpDown2].arrTargetPoint[4]:=arrAxisPar[AxiseNo.AxisName.CaCarryingUpDown2].arrTargetPoint[3]-arrAxisPar[AxiseNo.AxisName.CaCarryingUpDown2].arrTargetPoint[10];  //等待位置
//arrAxisPar[AxiseNo.AxisName.AnCarryingUpDown].arrTargetPoint[1]:=arrAxisPar[AxiseNo.AxisName.AnCarryingUpDown].arrTargetPoint[3]-arrAxisPar[AxiseNo.AxisName.AnCarryingUpDown].arrTargetPoint[11];  //安全位置

//负极送纠偏平台搬运升降取片凸轮创建 20240509 CF
fbCaCrectCamCarryingUpDown2(  //取片
	bCreatTable:=                         fbCaCrectCamCarryingUpDown2.bCreatTable , 
	Reset:=                                  stSysState.bReset  ,  
	iTable:=                                   TableNo.M_CaCarryingUpDown2   , 
	fMoveLength:=4, //取片高度
	fSaveLength:=arrAxisPar[AxiseNo.AxisName.CaCarryingUpDown2].arrTargetPoint[10] - arrAxisPar[AxiseNo.AxisName.CaCarryingUpDown2].arrTargetPoint[11],//安全高度
	//fInitLength:=arrAxisPar[AxiseNo.AxisName.CaCarryingUpDown2].arrTargetPoint[4],//升降轴耦合初始位
	fMasterKeyPos1:=110 , //
	fMasterKeyPos2:=250 , //144
	//fMasterKeyPos3:=240 , //198
	//fMasterKeyPos4:=310 , //324
	
    axisMaster:=                        arrAxis[AxiseNo.VirAxisName.VirMain] ,   
	axisSlave:=                           arrAxis[AxiseNo.AxisName.CaCarryingUpDown2] ,  

	bCreatTableDone=> , 
	bCreatTableError=> , 
	bError=> );
fbCaCrectCamCarryingUpDown2.bCreatTableDone;
fbCaCrectCamCarryingUpDown2.bCreatTableError;
fbCaCrectCamCarryingUpDown2.bError;


//负极送纠偏平台搬运升降放极片凸轮创建-
fbCaCrectCamCarryingUpDown2_1(   //--------放片
	bCreatTable:=                         fbCaCrectCamCarryingUpDown2_1.bCreatTable , 
	Reset:=                                  stSysState.bReset  ,  
	iTable:=                                   TableNo.M_CaCarryingUpDown2_1   , 
	fMoveLength:= arrAxisPar[AxiseNo.AxisName.CaCarryingUpDown2].arrTargetPoint[10]       ,//放片高度
	fSaveLength:=arrAxisPar[AxiseNo.AxisName.CaCarryingUpDown2].arrTargetPoint[10] - arrAxisPar[AxiseNo.AxisName.CaCarryingUpDown2].arrTargetPoint[11]  , //安全高度
	//fInitLength:=arrAxisPar[AxiseNo.AxisName.CaCarryingUpDown2].arrTargetPoint[4],//升降轴耦合初始位
	fMasterKeyPos1:=110 , //125
	fMasterKeyPos2:=250 , //
	fMasterKeyPos3:=260 , //
	fMasterKeyPos4:=320 , //
	fMasterKeyPos5:=359 , //
	//fMasterKeyPos6:=250 , //
	fSlaveVelo:=0.25 , //
	
    axisMaster:=                        arrAxis[AxiseNo.VirAxisName.VirMain] ,   
	axisSlave:=                           arrAxis[AxiseNo.AxisName.CaCarryingUpDown2] ,  

	bCreatTableDone=> , 
	bCreatTableError=> , 
	bError=> );
fbCaCrectCamCarryingUpDown2_1.bCreatTableDone;
fbCaCrectCamCarryingUpDown2_1.bCreatTableError;
fbCaCrectCamCarryingUpDown2_1.bError;

//负极送纠偏平台搬运升降放极片凸轮创建-
fbCaCrectCamCarryingUpDown2_3(   //--------放片
	bCreatTable:=                         fbCaCrectCamCarryingUpDown2_3.bCreatTable , 
	Reset:=                                   stSysState.bReset  ,  
	iTable:=                                  TableNo.M_CaCarryingUpDown2_3   , 
	//fMoveLength:= arrAxisPar[AxiseNo.AxisName.CaCarryingUpDown2].arrTargetPoint[10]       ,//放片高度
	fSaveLength:=arrAxisPar[AxiseNo.AxisName.CaCarryingUpDown2].arrTargetPoint[10] - arrAxisPar[AxiseNo.AxisName.CaCarryingUpDown2].arrTargetPoint[11]  , //安全高度
	//fInitLength:=arrAxisPar[AxiseNo.AxisName.CaCarryingUpDown2].arrTargetPoint[4],//升降轴耦合初始位
	fMasterKeyPos1:=110 , //130
	fMasterKeyPos2:=250 , //
	//fMasterKeyPos3:=260 , //
	//fMasterKeyPos4:=320 , //
	//fMasterKeyPos5:=359 , //
	//fMasterKeyPos6:=250 , //
	//fSlaveVelo:=0.25 , //
	
    axisMaster:=                        arrAxis[AxiseNo.VirAxisName.VirMain] ,   
	axisSlave:=                           arrAxis[AxiseNo.AxisName.CaCarryingUpDown2] ,  

	bCreatTableDone=> , 
	bCreatTableError=> , 
	bError=> );
fbCaCrectCamCarryingUpDown2_3.bCreatTableDone;
fbCaCrectCamCarryingUpDown2_3.bCreatTableError;
fbCaCrectCamCarryingUpDown2_3.bError;




//负极叠片搬运平移凸轮创建
fbCaCrectCamDTCarryingLine.fMoveLength:=ABS(arrAxisPar[AxiseNo.AxisName.CaDTCarryingLine].arrTargetPoint[1]- arrAxisPar[AxiseNo.AxisName.CaDTCarryingLine].arrTargetPoint[2]);
fbCaCrectCamDTCarryingLine(
	bCreatTable:=                fbCaCrectCamDTCarryingLine.bCreatTable , 
	Reset:=                          stSysState.bReset  ,  
	iTable:=                        TableNo.M_CaDTCarryingLine  , 
	fMoveLength:=              , 
	fMasterKeyPos:=          250 , //
	
	axisMaster:=                 arrAxis[AxiseNo.VirAxisName.VirMain] ,  
    axisSlave:=                    arrAxis[AxiseNo.AxisName.CaDTCarryingLine] ,  
	bCreatTableDone=> , 
	bCreatTableError=> , 
	bError=> );

fbCaCrectCamDTCarryingLine.bCreatTableDone;
fbCaCrectCamDTCarryingLine.bCreatTableError;
fbCaCrectCamDTCarryingLine.bError;



(**********20240528SJ***************)
arrAxisPar[AxiseNo.AxisName.CaDTCarryingUpDown].arrTargetPoint[10]:=6; //等待高度  参数可调
arrAxisPar[AxiseNo.AxisName.CaDTCarryingUpDown].arrTargetPoint[11]:=18; //抬升高度  参数可调
arrAxisPar[AxiseNo.AxisName.CaDTCarryingUpDown].arrTargetPoint[4]:=arrAxisPar[AxiseNo.AxisName.CaDTCarryingUpDown].arrTargetPoint[3]-arrAxisPar[AxiseNo.AxisName.CaDTCarryingUpDown].arrTargetPoint[10];  //等待位置    以放片位为基准
//arrAxisPar[AxiseNo.AxisName.AnDTCarryingUpDown].arrTargetPoint[1]:=arrAxisPar[AxiseNo.AxisName.AnDTCarryingUpDown].arrTargetPoint[3]-arrAxisPar[AxiseNo.AxisName.AnDTCarryingUpDown].arrTargetPoint[11];  //安全位置

//负极叠片搬运升降取片凸轮创建
fbCaCrectCamDTCarryingUpDown(//取片
	bCreatTable:=                         fbCaCrectCamDTCarryingUpDown.bCreatTable , 
	Reset:=                                  stSysState.bReset  ,  
	iTable:=                                   TableNo.M_CaDTCarryingUpDown   , 
	fMoveLength:=arrAxisPar[AxiseNo.AxisName.CaDTCarryingUpDown].arrTargetPoint[10]-(arrAxisPar[AxiseNo.AxisName.CaDTCarryingUpDown].arrTargetPoint[3]-arrAxisPar[AxiseNo.AxisName.CaDTCarryingUpDown].arrTargetPoint[2])               ,//取片高度
	fSaveLength:=arrAxisPar[AxiseNo.AxisName.CaDTCarryingUpDown].arrTargetPoint[10]-arrAxisPar[AxiseNo.AxisName.CaDTCarryingUpDown].arrTargetPoint[11]              , //安全位
	//fInitLength:=arrAxisPar[AxiseNo.AxisName.CaDTCarryingUpDown].arrTargetPoint[4],//升降轴耦合初始位
	fMasterKeyPos1:=125 , //
	fMasterKeyPos2:=250 , //
	fMasterKeyPos3:=260 , //
	fMasterKeyPos4:= 320, //
	fMasterKeyPos5:=359 , //
	fMasterKeyPos6:= , //
	fSlaveVelo:=0.25 , //
	
    axisMaster:=                        arrAxis[AxiseNo.VirAxisName.VirMain] ,   
	axisSlave:=                           arrAxis[AxiseNo.AxisName.CaDTCarryingUpDown] ,  

	bCreatTableDone=> , 
	bCreatTableError=> , 
	bError=> );
fbCaCrectCamDTCarryingUpDown.bCreatTableDone;
fbCaCrectCamDTCarryingUpDown.bCreatTableError;
fbCaCrectCamDTCarryingUpDown.bError;


//负极叠片搬运升降放片凸轮创建
IF  DP_Step0>3000 AND DP_Step0<=3080 THEN
     fbCaCrectCamDTCarryingUpDown1.iTableSel:=2;
ELSE	 
	 fbCaCrectCamDTCarryingUpDown1.iTableSel:=1;
END_IF		 

fbCaCrectCamDTCarryingUpDown1(//放片
	bCreatTable:=                         fbCaCrectCamDTCarryingUpDown1.bCreatTable , 
	Reset:=                                   stSysState.bReset  ,  
	iTable:=                                   TableNo.M_CaDTCarryingUpDown1   , 
	bCamIn:=  fbCaCamInDTCarryingUpDown.bCamInExecute AND  fbCaCamInDTCarryingUpDown.iTableSel=2    , 
	fMoveLength:=arrAxisPar[AxiseNo.AxisName.CaDTCarryingUpDown].arrTargetPoint[10] , //取片高度
	fSaveLength:=arrAxisPar[AxiseNo.AxisName.CaDTCarryingUpDown].arrTargetPoint[10]-arrAxisPar[AxiseNo.AxisName.CaDTCarryingUpDown].arrTargetPoint[11]  , //安全高度
	//fInitLength:=arrAxisPar[AxiseNo.AxisName.CaDTCarryingUpDown].arrTargetPoint[4] ,//升降轴耦合初始位
	fMasterKeyPos1:=120 , //208
	fMasterKeyPos2:=250 , //256
	fMasterKeyPos3:=260 , //256
	fMasterKeyPos4:=342 , //328
	fMasterKeyPos5:=359 , //328
	fSlaveVelo:=0.25 , //
    axisMaster:=                        arrAxis[AxiseNo.VirAxisName.VirMain] ,   
	axisSlave:=                           arrAxis[AxiseNo.AxisName.CaDTCarryingUpDown] ,  

	bCreatTableDone=> , 
	bCreatTableError=> , 
	bError=> );
fbCaCrectCamDTCarryingUpDown1.bCreatTableDone;
fbCaCrectCamDTCarryingUpDown1.bCreatTableError;
fbCaCrectCamDTCarryingUpDown1.bError;


//正极叠片搬运升降避让凸轮创建
fbCaCrectCamDTCarryingUpDown3(//放片
	bCreatTable:=fbCaCrectCamDTCarryingUpDown3.bCreatTable, 
	Reset:=stSysState.bReset  , 
	iTable:=TableNo.M_CaDTCarryingUpDown3 , 
	//fMoveLength:=arrAxisPar[AxiseNo.AxisName.AnDTCarryingUpDown].arrTargetPoint[10] ,//放片高度 
	fSaveLength:=arrAxisPar[AxiseNo.AxisName.CaDTCarryingUpDown].arrTargetPoint[10]-arrAxisPar[AxiseNo.AxisName.CaDTCarryingUpDown].arrTargetPoint[11]  , //安全高度
	//fInitLength:=arrAxisPar[AxiseNo.AxisName.AnDTCarryingUpDown].arrTargetPoint[4],//升降轴耦合初始位
	fMasterKeyPos1:=130 , //208
	fMasterKeyPos2:=260 , //256
	//fMasterKeyPos3:=260 , //256
	//fMasterKeyPos4:=342 , //328
//	fMasterKeyPos5:=359 , //328
//	fSlaveVelo:=0.25 , //
	axisSlave:=arrAxis[AxiseNo.AxisName.CaDTCarryingUpDown]  , 
	axisMaster:=arrAxis[AxiseNo.VirAxisName.VirMain]  , 
	bCreatTableDone=> , 
	bCreatTableError=> , 
	bError=> );
	
fbCaCrectCamDTCarryingUpDown3.bCreatTableDone;
fbCaCrectCamDTCarryingUpDown3.bCreatTableError;
fbCaCrectCamDTCarryingUpDown3.bError;











tCaCreate_TON(IN:= , PT:=T#0.5S , Q=> , ET=> );
IF Mach_Control.U.DT_iMode=3 OR Mach_Control.U.DT_iMode=0 THEN//在手动状态下
				//在触摸屏上生成凸轮
				//rCaCreate_TRIG(CLK:=Mach_Control.Ca_b.CreateCamStart , Q=> );	
				rCaCreate_TRIG(CLK:=(Mach_Control.Ca_b.CreateCamStart 
                                    AND	NOT arrAxisCtrl[AxiseNo.AxisName.CaCarryingLine2].Status.Coupled
									AND	NOT arrAxisCtrl[AxiseNo.AxisName.CaCarryingUpDown2].Status.Coupled
									AND	NOT arrAxisCtrl[AxiseNo.AxisName.CaDTCarryingLine].Status.Coupled
									AND	NOT arrAxisCtrl[AxiseNo.AxisName.CaDTCarryingUpDown].Status.Coupled), Q=> );				
				IF rCaCreate_TRIG.Q THEN
					tCaCreate_TON.IN:=FALSE;
					CaCrectCamStep0:=10;
					Mach_Control.Ca_b.Error[0]:=FALSE;
				END_IF
END_IF
				//负极取料凸轮自动创建
				CASE CaCrectCamStep0 OF
						10:
								IF NOT tCaCreate_TON.Q THEN
										//fbCaCrectCamCarryingLine1.bCreatTable :=TRUE;//负极取流水线平移凸轮创建
										//fbCaCrectCamCarryingUpDown1.bCreatTable:=TRUE;//负极取流水线放片升降凸轮创建
										//fbCaCrectCamCarryingUpDown1_1.bCreatTable:=TRUE;//负极取流水线取片升降凸轮创建
										//fbCaCrectCamCarryingWhirling.bCreatTable:=TRUE;//负极取流水线旋转凸轮创建
										 fbCaCrectCamCarryingLine2.bCreatTable :=FALSE;//负极送片搬运平移凸轮创建
										 fbCaCrectCamCarryingUpDown2.bCreatTable:=FALSE;//负极送片搬运升降取片凸轮创建
										 fbCaCrectCamCarryingUpDown2_1.bCreatTable:=FALSE;//负极送片搬运升降放片凸轮创建
										 fbCaCrectCamCarryingUpDown2_3.bCreatTable:=FALSE;//负极送片搬运升降放片凸轮创建
										 fbCaCrectCamDTCarryingLine.bCreatTable :=FALSE;//负极叠片搬运平移凸轮创建
										 fbCaCrectCamDTCarryingUpDown.bCreatTable:=FALSE;//负极叠片搬运升降取片凸轮创建
										 fbCaCrectCamDTCarryingUpDown1.bCreatTable:=FALSE;//负极叠片搬运升降放片凸轮创建
										  fbCaCrectCamDTCarryingUpDown3.bCreatTable:=FALSE;//负极叠片搬运升降放片凸轮创建
										 Mach_Control.Ca_b.CreateCamDone:=FALSE;
										 tCaCreate_TON.IN:=TRUE;					
								ELSE
											tCaCreate_TON.IN:=FALSE;	
											CaCrectCamStep0:=11;
								END_IF
								
						11:	
								IF  NOT Ca_Cam_ton[1].Q THEN
									arrAxisCtrl[AxiseNo.AxisName.CaCarryingLine2].Cmd.bStop:=TRUE;
									arrAxisCtrl[AxiseNo.AxisName.CaCarryingUpDown2].Cmd.bStop:=TRUE;
									arrAxisCtrl[AxiseNo.AxisName.CaDTCarryingLine].Cmd.bStop:=TRUE;
									arrAxisCtrl[AxiseNo.AxisName.CaDTCarryingUpDown].Cmd.bStop:=TRUE;
									Ca_Cam_ton[1].IN:=TRUE;
								ELSE
									Ca_Cam_ton[1].IN:=FALSE;
									CaCrectCamStep0:=12;
									arrAxisCtrl[AxiseNo.AxisName.CaCarryingLine2].Cmd.bStop:=FALSE;
									arrAxisCtrl[AxiseNo.AxisName.CaCarryingUpDown2].Cmd.bStop:=FALSE;
									arrAxisCtrl[AxiseNo.AxisName.CaDTCarryingLine].Cmd.bStop:=FALSE;
									arrAxisCtrl[AxiseNo.AxisName.CaDTCarryingUpDown].Cmd.bStop:=FALSE;
								END_IF
								
						12:
								IF  NOT Ca_Cam_ton[2].Q THEN
									arrAxisCtrl[AxiseNo.AxisName.CaCarryingLine2].Cmd.bReset:=TRUE;	
									arrAxisCtrl[AxiseNo.AxisName.CaCarryingUpDown2].Cmd.bReset:=TRUE;
									arrAxisCtrl[AxiseNo.AxisName.CaDTCarryingLine].Cmd.bReset:=TRUE;
									arrAxisCtrl[AxiseNo.AxisName.CaDTCarryingUpDown].Cmd.bReset:=TRUE;
									Ca_Cam_ton[2].IN:=TRUE;
								 ELSE
									 Ca_Cam_ton[2].IN:=FALSE;
									 CaCrectCamStep0:=13;
									arrAxisCtrl[AxiseNo.AxisName.CaCarryingLine2].Cmd.bReset:=FALSE;	
									arrAxisCtrl[AxiseNo.AxisName.CaCarryingUpDown2].Cmd.bReset:=FALSE;
									arrAxisCtrl[AxiseNo.AxisName.CaDTCarryingLine].Cmd.bReset:=FALSE;
									arrAxisCtrl[AxiseNo.AxisName.CaDTCarryingUpDown].Cmd.bReset:=FALSE;
								 END_IF
							

						13:
							arrAxisCtrl[AxiseNo.AxisName.CaCarryingLine2].Cmd.bEnable:=TRUE;
							arrAxisCtrl[AxiseNo.AxisName.CaCarryingUpDown2].Cmd.bEnable:=TRUE;
							arrAxisCtrl[AxiseNo.AxisName.CaDTCarryingLine].Cmd.bEnable:=TRUE;
							arrAxisCtrl[AxiseNo.AxisName.CaDTCarryingUpDown].Cmd.bEnable:=TRUE;
							IF arrAxisCtrl[AxiseNo.AxisName.CaCarryingLine2].Status.Enabled AND arrAxisCtrl[AxiseNo.AxisName.CaCarryingUpDown2].Status.Enabled AND
								arrAxisCtrl[AxiseNo.AxisName.CaDTCarryingLine].Status.Enabled AND arrAxisCtrl[AxiseNo.AxisName.CaDTCarryingUpDown].Status.Enabled THEN
								 CaCrectCamStep0:=20;
							END_IF
								
								
						20://凸轮创建
									//fbCaCrectCamCarryingLine1.bCreatTable :=TRUE;//负极取流水线平移凸轮创建
									//fbCaCrectCamCarryingUpDown1.bCreatTable:=TRUE;//负极取流水线放片升降凸轮创建
									//fbCaCrectCamCarryingUpDown1_1.bCreatTable:=TRUE;//负极取流水线取片升降凸轮创建
									//fbCaCrectCamCarryingWhirling.bCreatTable:=TRUE;//负极取流水线旋转凸轮创建
									 fbCaCrectCamCarryingLine2.bCreatTable :=TRUE;//负极送片搬运平移凸轮创建
									 fbCaCrectCamCarryingUpDown2.bCreatTable:=TRUE;//负极送片搬运升降取片凸轮创建
									 fbCaCrectCamCarryingUpDown2_1.bCreatTable:=TRUE;//负极送片搬运升降放片凸轮创建
									 fbCaCrectCamCarryingUpDown2_3.bCreatTable:=TRUE;//负极送片搬运升降放片凸轮创建
									 fbCaCrectCamDTCarryingLine.bCreatTable :=TRUE;//负极叠片搬运平移凸轮创建
									 fbCaCrectCamDTCarryingUpDown.bCreatTable:=TRUE;//负极叠片搬运升降取片凸轮创建
									 fbCaCrectCamDTCarryingUpDown1.bCreatTable:=TRUE;//负极叠片搬运升降放片凸轮创建
									  fbCaCrectCamDTCarryingUpDown3.bCreatTable:=TRUE;//负极叠片搬运升降放片凸轮创建
									 Mach_Control.Ca_b.CreateCamDone:=FALSE;
									 CaCrectCamStep0:=30;
						30://判断凸轮是否创建完成
									IF fbCaCrectCamCarryingLine2.bCreatTableDone AND  fbCaCrectCamCarryingUpDown2.bCreatTableDone AND  fbCaCrectCamCarryingUpDown2_1.bCreatTableDone  AND
										 fbCaCrectCamDTCarryingLine.bCreatTableDone AND fbCaCrectCamDTCarryingUpDown.bCreatTableDone AND fbCaCrectCamDTCarryingUpDown1.bCreatTableDone  AND
                                        fbCaCrectCamCarryingUpDown2_3.bCreatTableDone AND  fbCaCrectCamDTCarryingUpDown3.bCreatTableDone  THEN
											Mach_Control.Ca_b.CreateCamDone:=TRUE;
											CaCrectCamStep0:=6666;
									ELSE
											IF fbCaCrectCamCarryingLine2.bCreatTableError OR fbCaCrectCamCarryingUpDown2.bCreatTableError OR fbCaCrectCamCarryingUpDown2_1.bCreatTableError  OR 
												fbCaCrectCamDTCarryingLine.bCreatTableError OR fbCaCrectCamDTCarryingUpDown.bCreatTableError OR  fbCaCrectCamDTCarryingUpDown1.bCreatTableError OR 
                                          fbCaCrectCamCarryingUpDown2_3.bCreatTableError OR  fbCaCrectCamDTCarryingUpDown3.bCreatTableError    THEN								
												Mach_Control.Ca_b.Error[0]:=TRUE;//负极取片创建凸轮报警
												CaCrectCamStep0:=9999;
											END_IF
									END_IF
				END_CASE




(***********************************负极凸轮耦合***********************************************)
(*
      fbCaCamInCarryingLine1                      :FB_CamIn ;    
      fbCaCamInCarryingUpDown1               :FB_CamIn ;    
      fbCaCamInCarryingLine2                     :FB_CamIn ;    
      fbCaCamInCarryingUpDown2              :FB_CamIn ;    
      fbCaCamInDTCarryingLine                   :FB_CamIn ;    
      fbCaCamInDTCarryingUpDown            :FB_CamIn ;    
*)

//负极取流水线搬运平移凸轮耦合
fbCaCamInCarryingLine1.ParCamIn.SlaveScaling;
fbCaCamInCarryingLine1(
	Reset:=                      stSysState.bReset  , 
	bCamInExecute:=       fbCaCamInCarryingLine1.bCamInExecute, 
	iTable1:=                   TableNo.M_CaCarryingLine1  , 
	iTable2:=                   , 
	iTableSel:=                 , 
	ParCamIn:= , 
  	axisMaster:=            arrAxis[AxiseNo.VirAxisName.CaCarryingVirGM] ,  
	axisSlave:=               arrAxis[AxiseNo.AxisName.CaCarryingLine1] ,  
	bError=> , 
	bReady=> , 
	bInSync=> );

(*Mach_Control.Ca_b.Error[11]:=*)fbCaCamInCarryingLine1.bError;
fbCaCamInCarryingLine1.bReady;
fbCaCamInCarryingLine1.bInSync;

//负极取流水线搬运升降凸轮耦合
fbCaCamInCarryingUpDown1.iTableSel;
fbCaCamInCarryingUpDown1(
	Reset:=                      stSysState.bReset  , 
	bCamInExecute:=       fbCaCamInCarryingUpDown1.bCamInExecute, 
	iTable1:=                   TableNo.M_CaCarryingUpDown1  , 
	iTable2:=                   TableNo.M_CaCarryingUpDown1_1 , 
	iTableSel:=                  , 
	ParCamIn:=                  , 
  	axisMaster:=            arrAxis[AxiseNo.VirAxisName.CaCarryingVirGM] ,  
	axisSlave:=               arrAxis[AxiseNo.AxisName.CaCarryingUpDown1] ,  
	bError=> , 
	bReady=> , 
	bInSync=> );

(*Mach_Control.Ca_b.Error[12]:=*)fbCaCamInCarryingUpDown1.bError;
fbCaCamInCarryingUpDown1.bReady;
fbCaCamInCarryingUpDown1.bInSync;
//负极取流水线旋转
fbCaCamInCarryingWhirling.ParCamIn.SlaveScaling;
fbCaCamInCarryingWhirling(
	Reset:=                      stSysState.bReset  , 
	bCamInExecute:=       fbCaCamInCarryingWhirling.bCamInExecute, 
	iTable1:=                   TableNo.M_CaCarryingWhirling1  , 
	iTable2:=                   , 
	iTableSel:=                 , 
	ParCamIn:= , 
  	axisMaster:=            arrAxis[AxiseNo.VirAxisName.CaCarryingVirGM] ,  
	axisSlave:=               arrAxis[AxiseNo.AxisName.CaCarryingWhirling1] ,  
	bError=> , 
	bReady=> , 
	bInSync=> );

fbCaCamInCarryingWhirling.bError;
fbCaCamInCarryingWhirling.bReady;
fbCaCamInCarryingWhirling.bInSync;




//负极送片搬运平移凸轮耦合
fbCaCamInCarryingLine2.ParCamIn.SlaveScaling;
fbCaCamInCarryingLine2.ParCamIn.MasterScaling:=fCaScaling;//20240508 CF
fbCaCamInCarryingLine2(
	Reset:=                      stSysState.bReset  , 
	bCamInExecute:=       fbCaCamInCarryingLine2.bCamInExecute, 
	iTable1:=                   TableNo.M_CaCarryingLine2  , 
	iTable2:=                   , 
	iTableSel:=                 , 
	ParCamIn:= , 
  	axisMaster:=            arrAxis[AxiseNo.VirAxisName.VirMain] ,  
	axisSlave:=               arrAxis[AxiseNo.AxisName.CaCarryingLine2] ,  
	bError=> , 
	bReady=> , 
	bInSync=> );
(*Mach_Control.Ca_b.Error[13]:=*)fbCaCamInCarryingLine2.bError;
fbCaCamInCarryingLine2.bReady;
fbCaCamInCarryingLine2.bInSync;


//负极送纠偏搬动升降凸轮耦合
fbCaCamInCarryingUpDown2.ParCamIn.MasterScaling:=fCaScaling;//20240508 CF
fbCaCamInCarryingUpDown2(
	Reset:=                      stSysState.bReset  , 
	bCamInExecute:=       fbCaCamInCarryingUpDown2.bCamInExecute, 
	iTable1:=                   TableNo.M_CaCarryingUpDown2  , 
	iTable2:=                   TableNo.M_CaCarryingUpDown2_1  , 
	iTable3:=                   TableNo.M_CaCarryingUpDown2_3  , 
	iTableSel:=                  , //耦合凸轮选择
	ParCamIn:=                  , 
  	axisMaster:=            arrAxis[AxiseNo.VirAxisName.VirMain] ,  
	axisSlave:=               arrAxis[AxiseNo.AxisName.CaCarryingUpDown2] ,  
	bError=> , 
	bReady=> , 
	bInSync=> );

(*Mach_Control.Ca_b.Error[14]:=*)fbCaCamInCarryingUpDown2.bError;
fbCaCamInCarryingUpDown2.bReady;
fbCaCamInCarryingUpDown2.bInSync;


//负极叠台搬运平移凸轮耦合
fbCaCamInDTCarryingLine.ParCamIn.SlaveScaling;
fbCaCamInDTCarryingLine(
	Reset:=                      stSysState.bReset  , 
	bCamInExecute:=       fbCaCamInDTCarryingLine.bCamInExecute, 
	iTable1:=                   TableNo.M_CaDTCarryingLine  , 
	iTable2:=                   , 
	iTableSel:=                 , 
	ParCamIn:=                , 
  	axisMaster:=            arrAxis[AxiseNo.VirAxisName.VirMain] ,  
	axisSlave:=               arrAxis[AxiseNo.AxisName.CaDTCarryingLine] ,  
	bError=> , 
	bReady=> , 
	bInSync=> );
(*Mach_Control.Ca_b.Error[15]:=*)fbCaCamInDTCarryingLine.bError;
fbCaCamInDTCarryingLine.bReady;
fbCaCamInDTCarryingLine.bInSync;


//负极叠台搬运升降凸轮耦合
fbCaCamInDTCarryingUpDown(
	Reset:=                      stSysState.bReset  , 
	bCamInExecute:=       fbCaCamInDTCarryingUpDown.bCamInExecute, 
	iTable1:=                   TableNo.M_CaDTCarryingUpDown  , 
	iTable2:=                    TableNo.M_CaDTCarryingUpDown1, 
	iTable3:=                    TableNo.M_CaDTCarryingUpDown3, 
	iTableSel:=                  , 
	ParCamIn:=                  , 
  	axisMaster:=            arrAxis[AxiseNo.VirAxisName.VirMain] ,  
	axisSlave:=               arrAxis[AxiseNo.AxisName.CaDTCarryingUpDown] ,  
	bError=> , 
	bReady=> , 
	bInSync=> );

(*Mach_Control.Ca_b.Error[16]:=*)fbCaCamInDTCarryingUpDown.bError;
fbCaCamInDTCarryingUpDown.bReady;
fbCaCamInDTCarryingUpDown.bInSync;


IF fbCaCamInCarryingLine1.bError OR fbCaCamInCarryingUpDown1.bError OR fbCaCamInCarryingLine2.bError OR fbCaCamInCarryingUpDown2.bError OR fbCaCamInDTCarryingLine.bError OR fbCaCamInDTCarryingUpDown.bError THEN
		Mach_Control.Ca_b.Error[11]:=TRUE;//负极藕合凸轮报警
	ELSE	
		Mach_Control.Ca_b.Error[11]:=FALSE;
END_IF
END_ACTION

ACTION Ca_Conditions:
(********************负极放弃取片********************)
Mach_Control.Ca_b.JumpPiceReady:=Mach_Control.U.DT_iMode<>1 OR Mach_Control.Ca_b.Ca_SegbeltFalg OR Mach_Control.U.EmptyRunMode OR   (Mach_Control.DT_b.SinStepMode AND Ca_StandbyStep2<>35 AND Ca_StandbyStep2<>40);

(********************负极取片准备好********************)
Mach_Control.Ca_b.GetPiceReady:=NOT Mach_Control.Ca_b.JumpPiceReady AND
														arrAxisCtrl[AxiseNo.AxisName.CaCarryingUpDown1].Status.Homed AND arrAxisCtrl[AxiseNo.AxisName.CaCarryingUpDown1].Cmd.arrbRealPoint[1] AND
														arrAxisCtrl[AxiseNo.AxisName.CaCarryingLine1].Status.Homed AND arrAxisCtrl[AxiseNo.AxisName.CaCarryingLine1].Cmd.arrbRealPoint[1];
(*
IF Mach_Control.U.DT_iMode=1 AND NOT Mach_Control.Ca_b.Ca_SegbeltFalg AND (DP_Step0<>6030 AND DP_Step0<>6040 AND 
Mach_Control.An_b.An_Quantited <= Par.stDT_date.An_Quantity  AND  Mach_Control.Ca_b.Ca_Quantited < Par.stDT_date.Ca_Quantity) AND
   arrAxisCtrl[AxiseNo.AxisName.CaCarryingUpDown1].Status.Homed AND arrAxisCtrl[AxiseNo.AxisName.CaCarryingUpDown1].Cmd.arrbRealPoint[1] AND
   arrAxisCtrl[AxiseNo.AxisName.CaCarryingLine1].Status.Homed AND arrAxisCtrl[AxiseNo.AxisName.CaCarryingLine1].Cmd.arrbRealPoint[1] THEN
 		Mach_Control.Ca_b.GetPiceReady:=TRUE;
ELSE
 		Mach_Control.Ca_b.GetPiceReady:=FALSE;	
END_IF

IF Mach_Control.U.DT_iMode<>1 OR Mach_Control.Ca_b.Ca_SegbeltFalg OR JumpPiceReady_temp1 OR JumpPiceReady_temp2 OR JumpPiceReady_temp3 THEN
	Mach_Control.Ca_b.JumpPiceReady:=TRUE;
ELSE
	Mach_Control.Ca_b.JumpPiceReady:=FALSE;
END_IF
*)



//负极纠偏平台放极片允许
IF  NOT Mach_Control.Ca_b.Ca_deviationFalg AND arrAxisCtrl[AxiseNo.AxisName.CadeviationX1].Status.Homed AND NOT arrAxisCtrl[AxiseNo.AxisName.CadeviationX1].Status.Error AND 
	arrAxisCtrl[AxiseNo.AxisName.CadeviationX1].Status.NoMoving AND arrAxisCtrl[AxiseNo.AxisName.CadeviationX1].Cmd.arrbRealPoint[1] AND 
	arrAxisCtrl[AxiseNo.AxisName.CadeviationX2].Status.Homed AND NOT arrAxisCtrl[AxiseNo.AxisName.CadeviationX2].Status.Error AND 
	arrAxisCtrl[AxiseNo.AxisName.CadeviationX2].Status.NoMoving AND arrAxisCtrl[AxiseNo.AxisName.CadeviationX2].Cmd.arrbRealPoint[1] AND 
	arrAxisCtrl[AxiseNo.AxisName.CadeviationY].Status.Homed AND NOT arrAxisCtrl[AxiseNo.AxisName.CadeviationY].Status.Error AND 
	arrAxisCtrl[AxiseNo.AxisName.CadeviationY].Status.NoMoving AND arrAxisCtrl[AxiseNo.AxisName.CadeviationY].Cmd.arrbRealPoint[1] THEN
	Mach_Control.Ca_b.Ca_deviationFPOK:=TRUE;
ELSE
	Mach_Control.Ca_b.Ca_deviationFPOK:=FALSE;	
END_IF

//负极搬运皮带取极片允许
IF  Par.stDT_date.Ca_betlCount.5 AND arrAxisCtrl[AxiseNo.AxisName.CaBelt].Status.NoMoving AND NOT arrAxisCtrl[AxiseNo.AxisName.CaBelt].Status.Error THEN
	Mach_Control.Ca_b.Ca_CacheBeltDLOK:=TRUE;
ELSE
	Mach_Control.Ca_b.Ca_CacheBeltDLOK:=FALSE;	
END_IF



//负极搬运皮带放极片允许
IF NOT  Par.stDT_date.Ca_betlCount.0 AND arrAxisCtrl[AxiseNo.AxisName.CaCarryingUpDown1].Status.NoMoving AND NOT arrAxisCtrl[AxiseNo.AxisName.CaCarryingUpDown1].Status.Error  THEN
	Mach_Control.Ca_b.Ca_CacheBeltFLOK:=TRUE;
ELSE
	Mach_Control.Ca_b.Ca_CacheBeltFLOK:=FALSE;
END_IF
//负极搬运升降1、负极搬运升降2允许负极流水线电机转动   根据实际情况修改 20240509 CF
IF ((arrAxisCtrl[AxiseNo.AxisName.CaCarryingUpDown1].Status.fSetPos <= arrAxisPar[AxiseNo.AxisName.CaCarryingUpDown1].arrTargetPoint[3]-4
	  AND arrAxisCtrl[AxiseNo.AxisName.CaCarryingUpDown1].Status.Homed ) OR
	 (arrAxisCtrl[AxiseNo.AxisName.CaCarryingLine1].Status.fActPos < arrAxisPar[AxiseNo.AxisName.CaCarryingLine1].arrTargetPoint[2]-100  
	  AND arrAxisCtrl[AxiseNo.AxisName.CaCarryingLine1].Status.Homed ) ) AND
	 
	 ((arrAxisCtrl[AxiseNo.AxisName.CaCarryingUpDown2].Status.fSetPos <= arrAxisPar[AxiseNo.AxisName.CaCarryingUpDown2].arrTargetPoint[2]-4
	   AND arrAxisCtrl[AxiseNo.AxisName.CaCarryingUpDown2].Status.Homed ) OR 
	   (arrAxisCtrl[AxiseNo.AxisName.CaCarryingLine2].Status.fActPos > arrAxisPar[AxiseNo.AxisName.CaCarryingLine2].arrTargetPoint[1]+225  
	     AND  arrAxisCtrl[AxiseNo.AxisName.CaCarryingLine2].Status.Homed ) ) THEN
	Mach_Control.Ca_b.Ca_betlMoveOK:=TRUE;
ELSE
	Mach_Control.Ca_b.Ca_betlMoveOK:=FALSE;	
END_IF


(*  南昌备份
IF ((arrAxisCtrl[AxiseNo.AxisName.CaCarryingUpDown1].Status.fSetPos <= arrAxisPar[AxiseNo.AxisName.CaCarryingUpDown1].arrTargetPoint[1]+0.5)
	 OR arrAxisCtrl[AxiseNo.AxisName.CaCarryingLine1].Cmd.arrbRealPoint[1]) AND arrAxisCtrl[AxiseNo.AxisName.CaCarryingUpDown1].Status.Homed AND
	 
	 ((arrAxisCtrl[AxiseNo.AxisName.CaCarryingUpDown2].Status.fSetPos <= arrAxisPar[AxiseNo.AxisName.CaCarryingUpDown2].arrTargetPoint[4]+0.5) 
	OR arrAxisCtrl[AxiseNo.AxisName.CaCarryingLine2].Cmd.arrbRealPoint[2]) AND arrAxisCtrl[AxiseNo.AxisName.CaCarryingUpDown1].Status.Homed  THEN
	Mach_Control.Ca_b.Ca_betlMoveOK:=TRUE;
ELSE
	Mach_Control.Ca_b.Ca_betlMoveOK:=FALSE;	
END_IF
*)


//负极搬运平移2在安全位,、负极叠片升降在安全位、尾卷夹隔膜平移在安全位、允许负极叠片搬运平移移动纠偏平台位
//arrAxisCtrl[AxiseNo.AxisName.TailCurlSEPTALine].Status.Homed  AND arrAxisCtrl[AxiseNo.AxisName.TailCurlSEPTALine].Status.fActPos <= arrAxisPar[AxiseNo.AxisName.TailCurlSEPTALine].arrTargetPoint[1] 
IF arrAxisCtrl[AxiseNo.AxisName.CaCarryingLine2].Status.Homed AND arrAxisCtrl[AxiseNo.AxisName.CaCarryingLine2].Status.NoMoving AND arrAxisCtrl[AxiseNo.AxisName.CaCarryingLine2].Cmd.arrbRealPoint[1] AND
    arrAxisCtrl[AxiseNo.AxisName.CaDTCarryingUpDown].Status.Homed AND arrAxisCtrl[AxiseNo.AxisName.CaDTCarryingUpDown].Status.NoMoving AND  TailCurlSEPTA_SafePos AND
 	 arrAxisCtrl[AxiseNo.AxisName.CaDTCarryingUpDown].Status.fSetPos   <=arrAxisPar[AxiseNo.AxisName.CaDTCarryingUpDown].arrTargetPoint[4]+0.1 THEN
	Mach_Control.Ca_b.CarryingSafepos[0]:=TRUE;
ELSE
	Mach_Control.Ca_b.CarryingSafepos[0]:=FALSE;	
END_IF
//隔膜平移在正极片位、负极叠片搬运升降在安全位，允许负极叠片搬运平移至叠片位
IF arrAxisCtrl[AxiseNo.AxisName.SEPTATLine].Status.Homed  AND arrAxisCtrl[AxiseNo.AxisName.SEPTATLine].Status.NoMoving AND arrAxisCtrl[AxiseNo.AxisName.SEPTATLine].Cmd.arrbRealPoint[1] AND 
    arrAxisCtrl[AxiseNo.AxisName.CaDTCarryingUpDown].Status.Homed AND  arrAxisCtrl[AxiseNo.AxisName.CaDTCarryingUpDown].Status.NoMoving AND arrAxisCtrl[AxiseNo.AxisName.CaDTCarryingUpDown].Cmd.arrbRealPoint[1] AND
	arrAxis[AxiseNo.AxisName.TailCurlSEPTALine].Status.Homed  AND arrAxisCtrl[AxiseNo.AxisName.TailCurlSEPTALine].Status.fSetPos <= arrAxisPar[AxiseNo.AxisName.TailCurlSEPTALine].arrTargetPoint[1]   THEN
	Mach_Control.Ca_b.CarryingSafepos[1]:=TRUE;
ELSE
	Mach_Control.Ca_b.CarryingSafepos[1]:=FALSE;
END_IF
//负极送片搬运升降2在安全位，允许负极送片搬运2平移至取流水线极片位
IF arrAxisCtrl[AxiseNo.AxisName.CaCarryingUpDown2].Cmd.arrbRealPoint[1] AND arrAxisCtrl[AxiseNo.AxisName.CaCarryingLine2].Status.Homed AND
	arrAxisCtrl[AxiseNo.AxisName.CaCarryingLine2].Status.NoMoving THEN
	Mach_Control.Ca_b.CarryingSafepos[2]:=TRUE;
ELSE
	Mach_Control.Ca_b.CarryingSafepos[2]:=FALSE;
END_IF
//负极送片搬运升降2在安全位、负极叠片搬运在安全位，允许负极送片搬运2平移至纠偏位
IF arrAxisCtrl[AxiseNo.AxisName.CaCarryingUpDown2].Cmd.arrbRealPoint[1] AND arrAxisCtrl[AxiseNo.AxisName.CaCarryingUpDown2].Status.Homed AND
	arrAxisCtrl[AxiseNo.AxisName.CaCarryingUpDown2].Status.NoMoving AND arrAxisCtrl[AxiseNo.AxisName.CaDTCarryingLine].Status.Homed  AND 
	arrAxisCtrl[AxiseNo.AxisName.CaDTCarryingLine].Status.NoMoving AND arrAxisCtrl[AxiseNo.AxisName.CaDTCarryingLine].Cmd.arrbRealPoint[2]  THEN
	Mach_Control.Ca_b.CarryingSafepos[3]:=TRUE;
ELSE
	Mach_Control.Ca_b.CarryingSafepos[3]:=FALSE;
END_IF	
//负极送片搬运升降1在安全位，允许负极搬运平移1移动
IF  arrAxisCtrl[AxiseNo.AxisName.CaCarryingUpDown1].Cmd.arrbRealPoint[1] AND arrAxisCtrl[AxiseNo.AxisName.CaCarryingUpDown1].Status.Homed AND
	arrAxisCtrl[AxiseNo.AxisName.CaCarryingUpDown1].Status.NoMoving THEN
	Mach_Control.Ca_b.CarryingSafepos[4]:=TRUE;
ELSE
	Mach_Control.Ca_b.CarryingSafepos[4]:=FALSE;
END_IF		 
//负极送片搬运安全位，负极叠片搬运安全位，尾卷夹隔膜平移，允许纠偏平台移动
IF arrAxisCtrl[AxiseNo.AxisName.CaCarryingUpDown2].Status.Homed AND arrAxisCtrl[AxiseNo.AxisName.CaCarryingLine2].Status.Homed  AND 
	(arrAxisCtrl[AxiseNo.AxisName.CaCarryingUpDown2].Status.fSetPos<=(arrAxisPar[AxiseNo.AxisName.CaCarryingUpDown2].arrTargetPoint[4]+2) OR arrAxisCtrl[AxiseNo.AxisName.CaCarryingLine2].Cmd.arrbRealPoint[1]) AND 
    arrAxisCtrl[AxiseNo.AxisName.CaDTCarryingUpDown].Status.Homed AND arrAxisCtrl[AxiseNo.AxisName.CaDTCarryingLine].Status.Homed  AND 
	(arrAxisCtrl[AxiseNo.AxisName.CaDTCarryingUpDown].Status.fSetPos<=(arrAxisPar[AxiseNo.AxisName.CaDTCarryingUpDown].arrTargetPoint[4]+2) OR arrAxisCtrl[AxiseNo.AxisName.CaDTCarryingLine].Cmd.arrbRealPoint[2]) (*AND 
	arrAxisCtrl[AxiseNo.AxisName.TailCurlSEPTALine].Status.Homed AND arrAxisCtrl[AxiseNo.AxisName.TailCurlSEPTALine].Status.fActPos<=arrAxisPar[AxiseNo.AxisName.TailCurlSEPTALine].arrTargetPoint[1]  *) THEN
	Mach_Control.Ca_b.CarryingSafepos[5]:=TRUE;
ELSE
	Mach_Control.Ca_b.CarryingSafepos[5]:=FALSE;
END_IF		
//负极取流水线机械手在安全位，允许模切流水线移动
(*
IF arrAxisCtrl[AxiseNo.AxisName.CaCarryingUpDown1].Status.Homed AND NOT Mach_Control.Ca_b.Ca_MainBelting AND 
 	(arrAxisCtrl[AxiseNo.AxisName.CaCarryingUpDown1].Status.fSetPos<=arrAxisPar[AxiseNo.AxisName.CaCarryingUpDown1].arrTargetPoint[1]+0.2 OR 
	  arrAxisCtrl[AxiseNo.AxisName.CaCarryingLine1].Cmd.arrbRealPoint[1]	) THEN
	Mach_Control.Ca_b.Ca_BeltSafe:=TRUE;
ELSE
	Mach_Control.Ca_b.Ca_BeltSafe:=FALSE;
END_IF
*)
(*
IF  Mach_Control.Ca_b.Ca_MainBelting THEN
	Mach_Control.Ca_b.Ca_BeltSafe:=TRUE;
ELSIF NOT Mach_Control.Ca_b.Ca_MainBelting AND  arrAxisCtrl[AxiseNo.AxisName.CaCarryingUpDown1].Cmd.arrbRealPoint[4] THEN
	Mach_Control.Ca_b.Ca_BeltSafe:=FALSE;
END_IF
*)
IF  Mach_Control.Ca_b.Ca_MainBelting THEN
	Mach_Control.Ca_b.Ca_BeltSafe:=TRUE;
ELSE
	Mach_Control.Ca_b.Ca_BeltSafe:=FALSE;
END_IF
//负极主流水线取片完成延时复位
Ca_BeltTon(IN:=Mach_Control.Ca_b.Ca_BeltDone , PT:=T#20MS , Q=> , ET=> );
IF Ca_BeltTon.Q THEN
	Mach_Control.Ca_b.Ca_BeltDone:=FALSE;//复位主流水线取片完成
END_IF




/////////////////////////////////////////////////////////////
/////////////////////////////////////////////////////////
////////////////////////////////////////////电机条件

//负极送片皮带
IF Mach_Control.U.DT_iMode=3  AND arrAxisCtrl[AxiseNo.AxisName.CaCarryingUpDown1].Status.fActPos<= arrAxisPar[AxiseNo.AxisName.CaCarryingUpDown1].arrTargetPoint[1] +0.5
AND  arrAxisCtrl[AxiseNo.AxisName.CaCarryingUpDown2].Status.fActPos<=arrAxisPar[AxiseNo.AxisName.CaCarryingUpDown2].arrTargetPoint[4]+0.5  THEN
	arrAxisCtrl[AxiseNo.AxisName.CaBelt].Cmd.Home_Condition:=TRUE;
	arrAxisCtrl[AxiseNo.AxisName.CaBelt].Cmd.JogN_Condition:=TRUE;
	arrAxisCtrl[AxiseNo.AxisName.CaBelt].Cmd.JogP_Condition:=TRUE;
ELSE
	arrAxisCtrl[AxiseNo.AxisName.CaBelt].Cmd.Home_Condition:=FALSE;	
	arrAxisCtrl[AxiseNo.AxisName.CaBelt].Cmd.JogN_Condition:=FALSE;
	arrAxisCtrl[AxiseNo.AxisName.CaBelt].Cmd.JogP_Condition:=FALSE;
END_IF



//负极送片搬运1平移
IF Mach_Control.U.DT_iMode=3 AND arrAxisCtrl[AxiseNo.AxisName.CaCarryingUpDown1].Status.Homed AND
 	arrAxisCtrl[AxiseNo.AxisName.CaCarryingUpDown1].Status.fSetPos<= arrAxisPar[AxiseNo.AxisName.CaCarryingUpDown1].arrTargetPoint[1]+1 THEN
	arrAxisCtrl[AxiseNo.AxisName.CaCarryingLine1].Cmd.Home_Condition:=TRUE;
ELSE
arrAxisCtrl[AxiseNo.AxisName.CaCarryingLine1].Cmd.Home_Condition:=FALSE;	
END_IF

IF Mach_Control.U.DT_iMode=3 AND arrAxisCtrl[AxiseNo.AxisName.CaCarryingLine1].Status.Homed AND 
	arrAxisCtrl[AxiseNo.AxisName.CaCarryingUpDown1].Status.Homed AND
 	arrAxisCtrl[AxiseNo.AxisName.CaCarryingUpDown1].Status.fSetPos<= arrAxisPar[AxiseNo.AxisName.CaCarryingUpDown1].arrTargetPoint[1]+1 THEN
	arrAxisCtrl[AxiseNo.AxisName.CaCarryingLine1].Cmd.GoPoint_Condition[1]:=TRUE;
ELSE
	arrAxisCtrl[AxiseNo.AxisName.CaCarryingLine1].Cmd.GoPoint_Condition[1]:=FALSE;	
END_IF

IF Mach_Control.U.DT_iMode=3 AND arrAxisCtrl[AxiseNo.AxisName.CaCarryingLine1].Status.Homed AND
	arrAxisCtrl[AxiseNo.AxisName.CaCarryingUpDown1].Status.Homed AND
 	arrAxisCtrl[AxiseNo.AxisName.CaCarryingUpDown1].Status.fSetPos<= arrAxisPar[AxiseNo.AxisName.CaCarryingUpDown1].arrTargetPoint[1]+1 THEN
		arrAxisCtrl[AxiseNo.AxisName.CaCarryingLine1].Cmd.GoPoint_Condition[2]:=TRUE;
ELSE
		arrAxisCtrl[AxiseNo.AxisName.CaCarryingLine1].Cmd.GoPoint_Condition[2]:=FALSE;	
END_IF

//负极送片搬运1升降
IF Mach_Control.U.DT_iMode=3  THEN
	arrAxisCtrl[AxiseNo.AxisName.CaCarryingUpDown1].Cmd.Home_Condition:=TRUE;
ELSE
	arrAxisCtrl[AxiseNo.AxisName.CaCarryingUpDown1].Cmd.Home_Condition:=FALSE;	
END_IF

IF Mach_Control.U.DT_iMode=3 AND arrAxisCtrl[AxiseNo.AxisName.CaCarryingUpDown1].Status.Homed THEN
	arrAxisCtrl[AxiseNo.AxisName.CaCarryingUpDown1].Cmd.GoPoint_Condition[1]:=TRUE;
ELSE
	arrAxisCtrl[AxiseNo.AxisName.CaCarryingUpDown1].Cmd.GoPoint_Condition[1]:=FALSE;	
END_IF

IF arrAxisCtrl[AxiseNo.AxisName.CaCarryingLine1].Cmd.arrbRealPoint[1] AND  Mach_Control.U.DT_iMode=3 AND arrAxisCtrl[AxiseNo.AxisName.CaCarryingUpDown1].Status.Homed THEN
	arrAxisCtrl[AxiseNo.AxisName.CaCarryingUpDown1].Cmd.GoPoint_Condition[2]:=TRUE;
ELSE
	arrAxisCtrl[AxiseNo.AxisName.CaCarryingUpDown1].Cmd.GoPoint_Condition[2]:=FALSE;	
END_IF

IF arrAxisCtrl[AxiseNo.AxisName.CaCarryingLine1].Cmd.arrbRealPoint[2] AND  Mach_Control.U.DT_iMode=3 AND arrAxisCtrl[AxiseNo.AxisName.CaCarryingUpDown1].Status.Homed THEN
	arrAxisCtrl[AxiseNo.AxisName.CaCarryingUpDown1].Cmd.GoPoint_Condition[3]:=TRUE;
ELSE
	arrAxisCtrl[AxiseNo.AxisName.CaCarryingUpDown1].Cmd.GoPoint_Condition[3]:=FALSE;	
END_IF

//负极送片搬运2平移
IF Mach_Control.U.DT_iMode=3 AND arrAxisCtrl[AxiseNo.AxisName.CaCarryingUpDown2].Status.Homed AND
 arrAxisCtrl[AxiseNo.AxisName.CaCarryingUpDown2].Status.fSetPos<=arrAxisPar[AxiseNo.AxisName.CaCarryingUpDown2].arrTargetPoint[1]+1    AND
 arrCyCtrl[arrCyNo.CylinderName.CaScrapbinUDCy].Io.DIOFFSwitch  AND	 arrCyCtrl[arrCyNo.CylinderName.CaScrapbinCy].Io.DIOnSwitch  THEN
		arrAxisCtrl[AxiseNo.AxisName.CaCarryingLine2].Cmd.Home_Condition:=TRUE;
ELSE
		arrAxisCtrl[AxiseNo.AxisName.CaCarryingLine2].Cmd.Home_Condition:=FALSE;	
END_IF

IF Mach_Control.U.DT_iMode=3 AND arrAxisCtrl[AxiseNo.AxisName.CaCarryingUpDown2].Status.Homed AND
arrAxisCtrl[AxiseNo.AxisName.CaCarryingUpDown2].Status.fSetPos<=arrAxisPar[AxiseNo.AxisName.CaCarryingUpDown2].arrTargetPoint[1]+1 AND
 arrAxisCtrl[AxiseNo.AxisName.CaCarryingLine2].Status.Homed AND
  arrCyCtrl[arrCyNo.CylinderName.CaScrapbinUDCy].Io.DIOFFSwitch AND	 arrCyCtrl[arrCyNo.CylinderName.CaScrapbinCy].Io.DIOnSwitch   THEN
arrAxisCtrl[AxiseNo.AxisName.CaCarryingLine2].Cmd.GoPoint_Condition[1]:=TRUE;
ELSE
arrAxisCtrl[AxiseNo.AxisName.CaCarryingLine2].Cmd.GoPoint_Condition[1]:=FALSE;	
END_IF

IF  Mach_Control.U.DT_iMode=3 AND arrAxisCtrl[AxiseNo.AxisName.CaCarryingUpDown2].Status.Homed AND
	 arrAxisCtrl[AxiseNo.AxisName.CaCarryingUpDown2].Status.fSetPos<=arrAxisPar[AxiseNo.AxisName.CaCarryingUpDown2].arrTargetPoint[1]+1 AND
 	arrAxisCtrl[AxiseNo.AxisName.CaCarryingLine2].Status.Homed AND  arrAxisCtrl[AxiseNo.AxisName.CaDTCarryingLine].Cmd.arrbRealPoint[2] AND
    arrCyCtrl[arrCyNo.CylinderName.CaScrapbinUDCy].Io.DIOFFSwitch AND	 arrCyCtrl[arrCyNo.CylinderName.CaScrapbinCy].Io.DIOnSwitch   THEN

	arrAxisCtrl[AxiseNo.AxisName.CaCarryingLine2].Cmd.GoPoint_Condition[2]:=TRUE;
ELSE
	arrAxisCtrl[AxiseNo.AxisName.CaCarryingLine2].Cmd.GoPoint_Condition[2]:=FALSE;	
END_IF

//负极送片搬运2升降
IF Mach_Control.U.DT_iMode=3  THEN
	arrAxisCtrl[AxiseNo.AxisName.CaCarryingUpDown2].Cmd.Home_Condition:=TRUE;
ELSE
	arrAxisCtrl[AxiseNo.AxisName.CaCarryingUpDown2].Cmd.Home_Condition:=FALSE;	
END_IF

IF Mach_Control.U.DT_iMode=3 AND arrAxisCtrl[AxiseNo.AxisName.CaCarryingUpDown2].Status.Homed THEN
	arrAxisCtrl[AxiseNo.AxisName.CaCarryingUpDown2].Cmd.GoPoint_Condition[1]:=TRUE;
ELSE
	arrAxisCtrl[AxiseNo.AxisName.CaCarryingUpDown2].Cmd.GoPoint_Condition[1]:=FALSE;	
END_IF

IF (*arrAxisCtrl[AxiseNo.AxisName.CaCarryingLine2].Cmd.arrbRealPoint[1] AND*)  Mach_Control.U.DT_iMode=3 AND arrAxisCtrl[AxiseNo.AxisName.CaCarryingUpDown2].Status.Homed THEN
	arrAxisCtrl[AxiseNo.AxisName.CaCarryingUpDown2].Cmd.GoPoint_Condition[2]:=TRUE;
ELSE
	arrAxisCtrl[AxiseNo.AxisName.CaCarryingUpDown2].Cmd.GoPoint_Condition[2]:=FALSE;	
END_IF

IF (*arrAxisCtrl[AxiseNo.AxisName.CaCarryingLine2].Cmd.arrbRealPoint[2] AND*)  Mach_Control.U.DT_iMode=3 AND arrAxisCtrl[AxiseNo.AxisName.CaCarryingUpDown1].Status.Homed THEN
	arrAxisCtrl[AxiseNo.AxisName.CaCarryingUpDown2].Cmd.GoPoint_Condition[3]:=TRUE;
ELSE
	arrAxisCtrl[AxiseNo.AxisName.CaCarryingUpDown2].Cmd.GoPoint_Condition[3]:=FALSE;	
END_IF

IF (*arrAxisCtrl[AxiseNo.AxisName.CaCarryingLine2].Cmd.arrbRealPoint[1] AND*)  Mach_Control.U.DT_iMode=3 AND arrAxisCtrl[AxiseNo.AxisName.CaCarryingUpDown2].Status.Homed THEN
	arrAxisCtrl[AxiseNo.AxisName.CaCarryingUpDown2].Cmd.GoPoint_Condition[4]:=TRUE;
ELSE
	arrAxisCtrl[AxiseNo.AxisName.CaCarryingUpDown2].Cmd.GoPoint_Condition[4]:=FALSE;	
END_IF

IF (*arrAxisCtrl[AxiseNo.AxisName.CaCarryingLine2].Cmd.arrbRealPoint[1] AND*)  Mach_Control.U.DT_iMode=3 AND arrAxisCtrl[AxiseNo.AxisName.CaCarryingUpDown2].Status.Homed THEN
	arrAxisCtrl[AxiseNo.AxisName.CaCarryingUpDown2].Cmd.GoPoint_Condition[5]:=TRUE;
ELSE
	arrAxisCtrl[AxiseNo.AxisName.CaCarryingUpDown2].Cmd.GoPoint_Condition[5]:=FALSE;	
END_IF


//负极送片搬运1旋转
IF Mach_Control.U.DT_iMode=3  AND
	arrAxisCtrl[AxiseNo.AxisName.CaCarryingUpDown1].Status.fSetPos<=arrAxisPar[AxiseNo.AxisName.CaCarryingUpDown1].arrTargetPoint[1]  THEN
	arrAxisCtrl[AxiseNo.AxisName.CaCarryingWhirling1].Cmd.Home_Condition:=TRUE;
ELSE
	arrAxisCtrl[AxiseNo.AxisName.CaCarryingWhirling1].Cmd.Home_Condition:=FALSE;	
END_IF

IF Mach_Control.U.DT_iMode=3  AND arrAxisCtrl[AxiseNo.AxisName.CaCarryingUpDown1].Cmd.arrbRealPoint[1] AND arrAxisCtrl[AxiseNo.AxisName.CaCarryingWhirling1].Status.Homed THEN
	arrAxisCtrl[AxiseNo.AxisName.CaCarryingWhirling1].Cmd.GoPoint_Condition[1]:=TRUE;
ELSE
	arrAxisCtrl[AxiseNo.AxisName.CaCarryingWhirling1].Cmd.GoPoint_Condition[1]:=FALSE;	
END_IF

IF Mach_Control.U.DT_iMode=3  AND arrAxisCtrl[AxiseNo.AxisName.CaCarryingUpDown1].Cmd.arrbRealPoint[1] AND arrAxisCtrl[AxiseNo.AxisName.CaCarryingWhirling1].Status.Homed THEN
	arrAxisCtrl[AxiseNo.AxisName.CaCarryingWhirling1].Cmd.GoPoint_Condition[2]:=TRUE;
ELSE
	arrAxisCtrl[AxiseNo.AxisName.CaCarryingWhirling1].Cmd.GoPoint_Condition[2]:=FALSE;	
END_IF


//负极纠偏平台X1
IF Mach_Control.U.DT_iMode=3  OR  (DP_Step0>=6015 AND   DP_Step0<=6041)   THEN
	arrAxisCtrl[AxiseNo.AxisName.CadeviationX1].Cmd.Home_Condition:=TRUE;
ELSE
	arrAxisCtrl[AxiseNo.AxisName.CadeviationX1].Cmd.Home_Condition:=FALSE;	
END_IF

IF Mach_Control.U.DT_iMode=3 AND arrAxisCtrl[AxiseNo.AxisName.CadeviationX1].Status.Homed THEN
	arrAxisCtrl[AxiseNo.AxisName.CadeviationX1].Cmd.GoPoint_Condition[1]:=TRUE;
ELSE
	arrAxisCtrl[AxiseNo.AxisName.CadeviationX1].Cmd.GoPoint_Condition[1]:=FALSE;	
END_IF

IF Mach_Control.U.DT_iMode=3 AND arrAxisCtrl[AxiseNo.AxisName.CadeviationX1].Status.Homed THEN
	arrAxisCtrl[AxiseNo.AxisName.CadeviationX1].Cmd.GoPoint_Condition[2]:=TRUE;
ELSE
	arrAxisCtrl[AxiseNo.AxisName.CadeviationX1].Cmd.GoPoint_Condition[2]:=FALSE;	
END_IF

IF Mach_Control.U.DT_iMode=3 AND arrAxisCtrl[AxiseNo.AxisName.CadeviationX1].Status.Homed THEN
	arrAxisCtrl[AxiseNo.AxisName.CadeviationX1].Cmd.GoPoint_Condition[3]:=TRUE;
ELSE
	arrAxisCtrl[AxiseNo.AxisName.CadeviationX1].Cmd.GoPoint_Condition[3]:=FALSE;	
END_IF

IF Mach_Control.U.DT_iMode=3 AND arrAxisCtrl[AxiseNo.AxisName.CadeviationX1].Status.Homed THEN
	arrAxisCtrl[AxiseNo.AxisName.CadeviationX1].Cmd.GoPoint_Condition[4]:=TRUE;
ELSE
	arrAxisCtrl[AxiseNo.AxisName.CadeviationX1].Cmd.GoPoint_Condition[4]:=FALSE;	
END_IF

IF Mach_Control.U.DT_iMode=3 AND arrAxisCtrl[AxiseNo.AxisName.CadeviationX1].Status.Homed THEN
	arrAxisCtrl[AxiseNo.AxisName.CadeviationX1].Cmd.GoPoint_Condition[5]:=TRUE;
ELSE
	arrAxisCtrl[AxiseNo.AxisName.CadeviationX1].Cmd.GoPoint_Condition[5]:=FALSE;	
END_IF

//负极纠偏平台X2
IF Mach_Control.U.DT_iMode=3  OR  (DP_Step0>=6015 AND   DP_Step0<=6041)    THEN
	arrAxisCtrl[AxiseNo.AxisName.CadeviationX2].Cmd.Home_Condition:=TRUE;
ELSE
	arrAxisCtrl[AxiseNo.AxisName.CadeviationX2].Cmd.Home_Condition:=FALSE;	
END_IF

IF Mach_Control.U.DT_iMode=3 AND arrAxisCtrl[AxiseNo.AxisName.CadeviationX2].Status.Homed THEN
	arrAxisCtrl[AxiseNo.AxisName.CadeviationX2].Cmd.GoPoint_Condition[1]:=TRUE;
ELSE
	arrAxisCtrl[AxiseNo.AxisName.CadeviationX2].Cmd.GoPoint_Condition[1]:=FALSE;	
END_IF

IF Mach_Control.U.DT_iMode=3 AND arrAxisCtrl[AxiseNo.AxisName.CadeviationX2].Status.Homed THEN
	arrAxisCtrl[AxiseNo.AxisName.CadeviationX2].Cmd.GoPoint_Condition[2]:=TRUE;
ELSE
	arrAxisCtrl[AxiseNo.AxisName.CadeviationX2].Cmd.GoPoint_Condition[2]:=FALSE;	
END_IF

IF Mach_Control.U.DT_iMode=3 AND arrAxisCtrl[AxiseNo.AxisName.CadeviationX2].Status.Homed THEN
	arrAxisCtrl[AxiseNo.AxisName.CadeviationX2].Cmd.GoPoint_Condition[3]:=TRUE;
ELSE
	arrAxisCtrl[AxiseNo.AxisName.CadeviationX2].Cmd.GoPoint_Condition[3]:=FALSE;	
END_IF

IF Mach_Control.U.DT_iMode=3 AND arrAxisCtrl[AxiseNo.AxisName.CadeviationX2].Status.Homed THEN
	arrAxisCtrl[AxiseNo.AxisName.CadeviationX2].Cmd.GoPoint_Condition[4]:=TRUE;
ELSE
	arrAxisCtrl[AxiseNo.AxisName.CadeviationX2].Cmd.GoPoint_Condition[4]:=FALSE;	
END_IF

IF Mach_Control.U.DT_iMode=3 AND arrAxisCtrl[AxiseNo.AxisName.CadeviationX2].Status.Homed THEN
	arrAxisCtrl[AxiseNo.AxisName.CadeviationX2].Cmd.GoPoint_Condition[5]:=TRUE;
ELSE
	arrAxisCtrl[AxiseNo.AxisName.CadeviationX2].Cmd.GoPoint_Condition[5]:=FALSE;	
END_IF

//负极纠偏平台Y
IF Mach_Control.U.DT_iMode=3  OR  (DP_Step0>=6015 AND   DP_Step0<=6041)  THEN
	arrAxisCtrl[AxiseNo.AxisName.CadeviationY].Cmd.Home_Condition:=TRUE;
ELSE
	arrAxisCtrl[AxiseNo.AxisName.CadeviationY].Cmd.Home_Condition:=FALSE;	
END_IF

IF Mach_Control.U.DT_iMode=3 AND arrAxisCtrl[AxiseNo.AxisName.CadeviationY].Status.Homed THEN
	arrAxisCtrl[AxiseNo.AxisName.CadeviationY].Cmd.GoPoint_Condition[1]:=TRUE;
ELSE
	arrAxisCtrl[AxiseNo.AxisName.CadeviationY].Cmd.GoPoint_Condition[1]:=FALSE;	
END_IF

IF Mach_Control.U.DT_iMode=3 AND arrAxisCtrl[AxiseNo.AxisName.CadeviationY].Status.Homed THEN
	arrAxisCtrl[AxiseNo.AxisName.CadeviationY].Cmd.GoPoint_Condition[2]:=TRUE;
ELSE
	arrAxisCtrl[AxiseNo.AxisName.CadeviationY].Cmd.GoPoint_Condition[2]:=FALSE;	
END_IF

IF Mach_Control.U.DT_iMode=3 AND arrAxisCtrl[AxiseNo.AxisName.CadeviationY].Status.Homed THEN
	arrAxisCtrl[AxiseNo.AxisName.CadeviationY].Cmd.GoPoint_Condition[3]:=TRUE;
ELSE
	arrAxisCtrl[AxiseNo.AxisName.CadeviationY].Cmd.GoPoint_Condition[3]:=FALSE;	
END_IF

